# B&R Automation Studio project Soiled_PLC (part 3)

#### 7_sdc2Cyclic.ab
```automation-basic
PROGRAM _CYCLIC
	(* cyclic program *)

;Sequence 7 - Discharger 2 D[907]

;-----------------------------------------
;Revision 1.00 19/12/2005 D.J. First Issue
;-----------------------------------------

DischargerEnable 		= ((D[15] > 0) AND NOT Std.HaltSys)

;I_BagAtBuffer			= X[6].X07
I_OpenBag				= X[1].X05              ;CAN[2].DropLoad OR TestDrop
I_LoadDropped			= X[1].X06             ;CAN[2].LoadDropped OR TestDropped
I_BagAtBuffer			= X[1].X02 OR TestBuffer
I_BagAtDischarger		= X[1].X03 OR TestAtDisch
I_BagEmpty			  	= TRUE

I_BagAtEmptyBuffer		= FALSE ;X[6].X13
O_EmptyBagBufferOpen	= FALSE ;Y[6].Y13

O_BagReady				= FALSE
O_OpenBuffer 			= FALSE
O_Steadys				= FALSE
O_Closer				= FALSE
O_OpenBag				= FALSE
O_OpenStop				= FALSE

;Alarm
Alarm[10].Name 			= almNoAlarm ;Clear sequence alarm name
Alarm[10].Bag 			= 80
Alarm[10].Beacon		= TRUE
Alarm[10].Extra			= 0
Alarm[10].Time			= 3000

;Setup Sequence
STEP = D[910]
;Setup Pulse contact
PLS = (STEP <> LASTSTEP)
LASTSTEP = STEP

;Step 0 - Disabled
IF (STEP = 0) THEN
	;Disabled
ENDIF

;Check Status - Bag settled at buffer, no bag at discharger, bag at buffer on screen and no bag at discharger on the screen
TON_10ms(I_BagAtBuffer,300,SettledAtBuffer,SettledAtBufferET)
IF (STEP = 1) THEN
	IF (NOT I_BagAtDischarger AND  (Bag[80].Cat = 0) AND NOT Std.HaltSys AND DischargerEnable AND SettledAtBuffer) THEN
		Request.DC[2] = TRUE
		D[910] = 2
	ENDIF
	IF I_BagAtDischarger THEN
		;D[907] = 2
	ENDIF
	IF (Bag[80].Cat > 0) THEN
		Alarm[10].Name = almBagDataError
	ELSE IF I_BagAtDischarger THEN
		Alarm[10].Name = almSwitchFault
	ELSE IF (Bag[80].Cat > 0) AND NOT I_BagAtBuffer THEN
		Alarm[10].Name 	= almBagNotAtProx
		Alarm[10].Bag	= 80
	ELSE IF (Bag[80].Cat = 0) AND I_BagAtBuffer AND DischargerEnable  THEN
		Alarm[10].Name 	= almBagNotShownOnScreen
		Alarm[10].Bag	= 80
	ENDIF
ENDIF

;Wait for bag in discharger
IF (STEP = 2) THEN
	O_OpenBuffer 	= TRUE
	IF I_BagAtDischarger THEN
		D[910] = 3
	ENDIF
	Alarm[10].Name = almNoAlarm ;almBagNotArrived
ENDIF

;Let bag settle in discharger
TON_10ms(((STEP = 3) AND I_BagAtDischarger),1000,SettledAtDischarger,SettledAtDischargerET)
IF (STEP = 3) THEN
	IF (Bag[80].Cat = 0) AND (Bag[81].Cat > 0) THEN
		Bag[80] = Bag[81]
		Bag[81] = Bag[0]
	ENDIF
	IF SettledAtDischarger THEN
		D[910] = 4
	ENDIF
	Alarm[10].Name = almBagNotSettled
ENDIF

;Allow steadys to move down
TON_10ms((STEP = 4),400,SteadysDown,SteadysDownET)
IF (STEP = 4) THEN
	IF SteadysDown THEN
		D[910] = 5
	ENDIF
	IF (Bag[80].Cat = Std.MaxCats) THEN
		D[910] = 8
	ENDIF
ENDIF

;Steady cylinders on from steps 4 - 9
O_Steadys = ((STEP >= 4) AND (STEP <= 9))

;Bag opener on from step 5 - 8
O_OpenBag = ((STEP >= 6) AND (STEP <= 8))

CodeStep  = ((STEP >= 4) AND (STEP <= 5))

;Wash Codes
IF CodeStep THEN

	Weight = Bag[80].Wgt

	;round up weight to give to wash machine
	Remainder = SINT(Bag[80].Wgt MOD 10)
	IF (Remainder > 4) THEN
		WgtRound = (Weight + 10)
	ELSE
		WgtRound = Weight
	ENDIF
ELSE
ENDIF

;Bag Ready to Washing Machine
IF (STEP = 5) THEN
	O_BagReady = TRUE

	IF I_OpenBag OR TestDischarger THEN
		D[910] = 6
	ENDIF
ELSE

ENDIF

;Set LoadDropped to False
IF (STEP <> 6) THEN
	LoadDropped = FALSE
ENDIF

;Open Bag Until LoadDropped recieved and has been open for 6 seconds
TON_10ms((STEP = 6),600,MinOpen,MinOpenET) ;ET means Elapsed Time
TON_10ms((STEP = 6) AND NOT I_DischargerBagEmpty ,100,BagEmpty,BagEmptyET)

IF (STEP = 6) THEN

	;IF I_LoadDropped  OR TestDischarger THEN

		LoadDropped = TRUE
	;ENDIF

	IF (LoadDropped AND MinOpen) THEN
		;Write Report
		;------------

	ENDIF
	IF (LoadDropped AND MinOpen ) THEN
		IF (ReportUnloading[5].Cat = 0) THEN
			ReportUnloading[5].Cat = UINT(Bag[80].Cat)	;Category
			ReportUnloading[5].Cus = Bag[80].Cus		;Customer
			ReportUnloading[5].Wgt = Bag[80].Wgt		;Weight
			ReportUnloading[5].Cnt = 0					;Count
			ReportUnloading[5].Stn = 0					;Station
			ReportUnloading[5].Mcn = 5					;Machine
		ENDIF
		D[910] = 7
	ENDIF
	Alarm[10].Time			= 600
	Alarm[10].Name = almLoadNotDropped
	ELSE
	LoadDropped = FALSE
ENDIF

;Change display to empty bag
IF (STEP = 7) THEN
	IF ((NOT I_OpenBag  AND I_BagEmpty) OR TestDrop) THEN
		Bag[80].Prg 	= Std.MaxProg
		Bag[80].Cat 	= Std.MaxCats
		Bag[80].Cus 	= Std.MaxCust

		D[910] 			= 8
	ENDIF
	Alarm[10].Name = almGeneralSequence
ENDIF

;Allow steadys to go up
TON_10ms((STEP = 8),400,SteadyUp,SteadyUpET)
IF (STEP = 8) THEN
	IF SteadyUp THEN
		D[910] = 9
	ENDIF
ENDIF

;Request empty bag release
IF (STEP = 9) THEN

	IF Line[32].Clear THEN
		C[32]  = 0
		D[910] = 10
	ENDIF
ENDIF

;Open buffer stop - unitl bag out
IF (STEP = 10) THEN
	O_OpenStop = TRUE
	Bag[80].Cat = 0
	Bag[80].Cus = 0
	Bag[80].Wgt = 0
	IF Line[32].Trip THEN
		D[910] = 1
	ENDIF
	Alarm[10].Name = almBagNotReleased
ENDIF

;Alarms
TimerAlarm.IN 	= NOT PLS AND (Alarm[10].Name > 0)
TimerAlarm.PT 	= Alarm[10].Time
TimerAlarm FUB TON_10ms()
Alarm[10].On 	= TimerAlarm.Q
Alarm[10].ET 	= TimerAlarm.ET

;Outputs
Y[1].Y02 = O_OpenBuffer
Y[1].Y04= O_Steadys
Y[1].Y06 = O_OpenBag
Y[1].Y03 = O_OpenStop
Y[1].Y05 = O_BagReady
END_PROGRAM
```

### Program Logical/Sequences/10ms/11_sdc6 (IEC) - * SDC2 Machine 2 CAN

#### 7_sdc2Cyclic.ab
```automation-basic
PROGRAM _CYCLIC
	(* cyclic program *)

;Sequence 7 - Discharger 2 D[907]

;-----------------------------------------
;Revision 1.00 19/12/2005 D.J. First Issue
;-----------------------------------------

DischargerEnable 		= ((D[26] > 0) AND NOT Std.HaltSys)

;I_BagAtBuffer			= X[6].X07
I_OpenBag				= X[1].X11
I_LoadDropped			= X[1].X12
I_BagAtBuffer			= X[1].X08 OR TestBuffer
I_BagAtDischarger		= X[1].X09 OR TestAtDisch
I_BagEmpty			  	= TRUE
I_BagOut                  = X[1].X10

RequestRel.DC[6]                   = FALSE

O_BagReady				= FALSE
O_OpenBuffer 			= FALSE
O_Steadys				= FALSE
O_Closer				= FALSE
O_OpenBag				= FALSE
O_OpenStop				= FALSE

;Alarm
Alarm[11].Name 			= almNoAlarm ;Clear sequence alarm name
Alarm[11].Bag 			= 85
Alarm[11].Beacon			= TRUE
Alarm[11].Extra			= 0
Alarm[11].Time			= 3000

;Setup Sequence
STEP = D[911]
;Setup Pulse contact
PLS = (STEP <> LASTSTEP)
LASTSTEP = STEP

;Step 0 - Disabled
IF (STEP = 0) THEN
	;Disabled
ENDIF

;Check Status - Bag settled at buffer, no bag at discharger, bag at buffer on screen and no bag at discharger on the screen
TON_10ms(I_BagAtBuffer,300,SettledAtBuffer,SettledAtBufferET)
IF (STEP = 1) THEN
	IF (NOT I_BagAtDischarger AND  (Bag[85].Cat = 0) AND NOT Std.HaltSys AND DischargerEnable AND SettledAtBuffer) THEN

		D[911] = 2
	ENDIF
	IF I_BagAtDischarger THEN
		;D[907] = 2
	ENDIF
	IF (Bag[85].Cat > 0) THEN
		Alarm[11].Name = almBagDataError
	ELSE IF I_BagAtDischarger THEN
		Alarm[11].Name = almSwitchFault
	ELSE IF (Bag[85].Cat > 0) AND NOT I_BagAtBuffer THEN
		Alarm[11].Name 	= almBagNotAtProx
		Alarm[11].Bag	= 85
	ELSE IF (Bag[85].Cat = 0) AND I_BagAtBuffer AND DischargerEnable  THEN
		Alarm[11].Name 	= almBagNotShownOnScreen
		Alarm[11].Bag	= 85
	ENDIF
ENDIF

;Wait for bag in discharger
IF (STEP = 2) THEN
	O_OpenBuffer 	= TRUE
	IF I_BagAtDischarger THEN
		D[911] = 3
	ENDIF
	Alarm[11].Name = almNoAlarm ;almBagNotArrived
ENDIF

;Let bag settle in discharger
TON_10ms(((STEP = 3) AND I_BagAtDischarger),1000,SettledAtDischarger,SettledAtDischargerET)
IF (STEP = 3) THEN
	IF (Bag[85].Cat = 0) AND (Bag[86].Cat > 0) THEN
		Bag[85] = Bag[86]
		Bag[86] = Bag[0]
	ENDIF
	IF SettledAtDischarger THEN
		D[911] = 4
	ENDIF
	Alarm[11].Name = almBagNotSettled
ENDIF

;Allow steadys to move down
TON_10ms((STEP = 4),400,SteadysDown,SteadysDownET)
IF (STEP = 4) THEN
	IF SteadysDown THEN
		D[911] = 5
	ENDIF
	IF (Bag[85].Cat = Std.MaxCats) THEN
		D[911] = 8
	ENDIF
ENDIF

;Steady cylinders on from steps 4 - 9
O_Steadys = ((STEP >= 4) AND (STEP <= 7))

;Bag opener on from step 5 - 8
O_OpenBag = ((STEP >= 6) AND (STEP <= 7))

CodeStep  = ((STEP >= 4) AND (STEP <= 5))

;Wash Codes
IF CodeStep THEN

	Weight = Bag[85].Wgt

	;round up weight to give to wash machine
	Remainder = SINT(Bag[85].Wgt MOD 10)
	IF (Remainder > 4) THEN
		WgtRound = (Weight + 10)
	ELSE
		WgtRound = Weight
	ENDIF

	;WashCodes
	;if Below the Machine limit of 99 and no WashCode has been entered then send the Category

ELSE

ENDIF

;Bag Ready to Washing Machine
IF (STEP = 5) THEN
	O_BagReady		= TRUE

	IF I_OpenBag OR TestDischarger THEN
		D[911] = 6
	ENDIF
ELSE
	O_BagReady		= FALSE
ENDIF

;Set LoadDropped to False
IF (STEP <> 6) THEN
	LoadDropped = FALSE
ENDIF

;Open Bag Until LoadDropped recieved and has been open for 6 seconds
TON_10ms((STEP = 6),600,MinOpen,MinOpenET) ;ET means Elapsed Time
TON_10ms((STEP = 6) AND NOT I_DischargerBagEmpty ,100,BagEmpty,BagEmptyET)

IF (STEP = 6) THEN

	IF I_LoadDropped  OR TestDischarger THEN

		LoadDropped = TRUE
	ENDIF

	IF (LoadDropped AND MinOpen) THEN
		;Write Report
		;------------

	ENDIF
	IF (LoadDropped AND MinOpen ) THEN
		IF (ReportUnloading[6].Cat = 0) THEN
			ReportUnloading[6].Cat = UINT(Bag[85].Cat)	;Category
			ReportUnloading[6].Cus = Bag[85].Cus		;Customer
			ReportUnloading[6].Wgt = Bag[85].Wgt		;Weight
			ReportUnloading[6].Cnt = 0					;Count
			ReportUnloading[6].Stn = 0					;Station
			ReportUnloading[6].Mcn = 6					;Machine
		ENDIF
		D[911] = 7
	ENDIF
	Alarm[11].Time			= 600
	Alarm[11].Name = almLoadNotDropped
	ELSE
	LoadDropped = FALSE
ENDIF

;Change display to empty bag
IF (STEP = 7) THEN
	IF ((NOT I_OpenBag  AND I_BagEmpty) OR TestDrop) THEN
		Bag[85].Prg 	= Std.MaxProg
		Bag[85].Cat 	= Std.MaxCats
		Bag[85].Cus 	= Std.MaxCust

		D[911] 			= 8
	ENDIF
	Alarm[11].Name = almGeneralSequence
ENDIF

;Allow steadys to go up
TON_10ms((STEP = 8),400,SteadyUp,SteadyUpET)
IF (STEP = 8) THEN
	IF SteadyUp THEN
		D[911] = 9
	ENDIF
ENDIF

;Request empty bag release
IF (STEP = 9) THEN
	RequestRel.DC[6] = TRUE
	IF Enable.DCEmptyRelease[6] THEN
		;C[32]  = 0
		D[911] = 10
	ENDIF
ENDIF

;Open buffer stop - unitl bag out
IF (STEP = 10) THEN
	O_OpenStop = TRUE
	Bag[85].Cat = 0
	Bag[85].Cus = 0
	Bag[85].Wgt = 0
	IF NOT Enable.DCEmptyRelease[6] OR I_BagOut THEN
		D[911] = 1
	ENDIF
	Alarm[11].Name = almBagNotReleased
ENDIF

;Alarms
TimerAlarm.IN 	= NOT PLS AND (Alarm[11].Name > 0)
TimerAlarm.PT 	= Alarm[11].Time
TimerAlarm FUB TON_10ms()
Alarm[11].On 	= TimerAlarm.Q
Alarm[11].ET 	= TimerAlarm.ET

;Outputs
Y[1].Y08 = O_OpenBuffer
Y[1].Y10 = O_Steadys
Y[1].Y12 = O_OpenBag
Y[1].Y09 = O_OpenStop
Y[1].Y11 = O_BagReady
END_PROGRAM
```

### Program Logical/Sequences/10ms/12_sdc7 (IEC) - * SDC2 Machine 2 CAN

#### 7_sdc2Cyclic.ab
```automation-basic
PROGRAM _CYCLIC
	(* cyclic program *)

;Sequence 7 - Discharger 2 D[907]

;-----------------------------------------
;Revision 1.00 19/12/2005 D.J. First Issue
;-----------------------------------------

DischargerEnable 		= ((D[27] > 0) AND NOT Std.HaltSys)

;I_BagAtBuffer			= X[6].X07
I_OpenBag				= X[2].X01 ;0CAN[2].DropLoad OR TestDrop
I_LoadDropped			= X[2].X02
I_BagAtBuffer			= X[1].X14 OR TestBuffer
I_BagAtDischarger		= X[1].X15 OR TestAtDisch
I_BagEmpty			  	= TRUE
I_BagOut                  = X[1].X16

I_BagAtEmptyBuffer		= FALSE ;X[6].X13
O_EmptyBagBufferOpen	= FALSE ;Y[6].Y13

O_BagReady				= FALSE
O_OpenBuffer 			= FALSE
O_Steadys				= FALSE
O_Closer				= FALSE
O_OpenBag				= FALSE
O_OpenStop				= FALSE

;Alarm
Alarm[12].Name 			= almNoAlarm ;Clear sequence alarm name
Alarm[12].Bag 			= 90
Alarm[12].Beacon		= TRUE
Alarm[12].Extra			= 0
Alarm[12].Time			= 3000

;Setup Sequence
STEP = D[912]
;Setup Pulse contact
PLS = (STEP <> LASTSTEP)
LASTSTEP = STEP

;Step 0 - Disabled
IF (STEP = 0) THEN
	;Disabled
ENDIF

;Check Status - Bag settled at buffer, no bag at discharger, bag at buffer on screen and no bag at discharger on the screen
TON_10ms(I_BagAtBuffer,300,SettledAtBuffer,SettledAtBufferET)
IF (STEP = 1) THEN
	IF (NOT I_BagAtDischarger AND  (Bag[90].Cat = 0) AND NOT Std.HaltSys AND DischargerEnable AND SettledAtBuffer) THEN

		D[912] = 2
	ENDIF
	IF I_BagAtDischarger THEN
		;D[907] = 2
	ENDIF
	IF (Bag[90].Cat > 0) THEN
		Alarm[12].Name = almBagDataError
	ELSE IF I_BagAtDischarger THEN
		Alarm[12].Name = almSwitchFault
	ELSE IF (Bag[91].Cat > 0) AND NOT I_BagAtBuffer THEN
		Alarm[12].Name 	= almBagNotAtProx
		Alarm[12].Bag	= 91
	ELSE IF (Bag[91].Cat = 0) AND I_BagAtBuffer AND DischargerEnable  THEN
		Alarm[12].Name 	= almBagNotShownOnScreen
		Alarm[12].Bag	= 91
	ENDIF
ENDIF

;Wait for bag in discharger
IF (STEP = 2) THEN
	O_OpenBuffer 	= TRUE
	IF I_BagAtDischarger THEN
		D[912] = 3
	ENDIF
	Alarm[12].Name = almNoAlarm ;almBagNotArrived
ENDIF

;Let bag settle in discharger
TON_10ms(((STEP = 3) AND I_BagAtDischarger),1000,SettledAtDischarger,SettledAtDischargerET)
IF (STEP = 3) THEN
	IF (Bag[90].Cat = 0) AND (Bag[91].Cat > 0) THEN
		Bag[90] = Bag[91]
		Bag[91] = Bag[0]
	ENDIF
	IF SettledAtDischarger THEN
		D[912] = 4
	ENDIF
	Alarm[12].Name = almBagNotSettled
ENDIF

;Allow steadys to move down
TON_10ms((STEP = 4),400,SteadysDown,SteadysDownET)
IF (STEP = 4) THEN
	IF SteadysDown THEN
		D[912] = 5
	ENDIF
	IF (Bag[90].Cat = Std.MaxCats) THEN
		D[912] = 8
	ENDIF
ENDIF

;Steady cylinders on from steps 4 - 9
O_Steadys = ((STEP >= 4) AND (STEP <= 9))

;Bag opener on from step 5 - 8
O_OpenBag = ((STEP >= 6) AND (STEP <= 8))

CodeStep  = ((STEP >= 4) AND (STEP <= 5))

;Wash Codes
IF CodeStep THEN

	Weight = Bag[90].Wgt

	;round up weight to give to wash machine
	Remainder = SINT(Bag[90].Wgt MOD 10)
	IF (Remainder > 4) THEN
		WgtRound = (Weight + 10)
	ELSE
		WgtRound = Weight
	ENDIF

ELSE

ENDIF

;Bag Ready to Washing Machine
IF (STEP = 5) THEN
	O_BagReady 		= TRUE

	IF I_OpenBag OR TestDischarger THEN
		D[912] = 6
	ENDIF
ELSE

ENDIF

;Set LoadDropped to False
IF (STEP <> 6) THEN
	LoadDropped = FALSE
ENDIF

;Open Bag Until LoadDropped recieved and has been open for 6 seconds
TON_10ms((STEP = 6),600,MinOpen,MinOpenET) ;ET means Elapsed Time
TON_10ms((STEP = 6) AND NOT I_DischargerBagEmpty ,100,BagEmpty,BagEmptyET)

IF (STEP = 6) THEN

	;IF I_LoadDropped  OR TestDischarger THEN

		LoadDropped = TRUE
	;ENDIF

	IF (LoadDropped AND MinOpen) THEN
		;Write Report
		;------------

	ENDIF
	IF (LoadDropped AND MinOpen ) THEN
		IF (ReportUnloading[2].Cat = 0) THEN
			ReportUnloading[2].Cat = UINT(Bag[90].Cat)	;Category
			ReportUnloading[2].Cus = Bag[90].Cus		;Customer
			ReportUnloading[2].Wgt = Bag[90].Wgt		;Weight
			ReportUnloading[2].Cnt = 0					;Count
			ReportUnloading[2].Stn = 0					;Station
			ReportUnloading[2].Mcn = 7					;Machine
		ENDIF
		D[912] = 7
	ENDIF
	Alarm[12].Time			= 600
	Alarm[12].Name = almLoadNotDropped
	ELSE
	LoadDropped = FALSE
ENDIF

;Change display to empty bag
IF (STEP = 7) THEN
	IF ((NOT I_OpenBag  AND I_BagEmpty) OR TestDrop) THEN
		Bag[90].Prg 	= Std.MaxProg
		Bag[90].Cat 	= Std.MaxCats
		Bag[90].Cus 	= Std.MaxCust

		D[912] 			= 8
	ENDIF
	Alarm[12].Name = almGeneralSequence
ENDIF

;Allow steadys to go up
TON_10ms((STEP = 8),400,SteadyUp,SteadyUpET)
IF (STEP = 8) THEN
	IF SteadyUp AND NOT Enable.DCEmptyRelease[7] THEN
		D[912] = 9
	ENDIF
	IF Enable.DCEmptyRelease[7]  THEN
		Alarm[12].Time			= 600
		Alarm[12].Name = almSwitchFault
	ENDIF
ENDIF

;Request empty bag release
IF (STEP = 9) THEN
	RequestRel.DC[7] = TRUE
	IF Enable.DCEmptyRelease[7] THEN
		;C[32]  = 0
		D[912] = 10
	ENDIF
	ELSE
	RequestRel.DC[7] = FALSE
ENDIF

;Open buffer stop - unitl bag out
IF (STEP = 10) THEN
	O_OpenStop = TRUE
	Bag[90].Cat = 0
	Bag[90].Cus = 0
	Bag[90].Wgt = 0
	IF NOT Enable.DCEmptyRelease[7]  OR I_BagOut THEN
		D[912] = 1
	ENDIF
	Alarm[12].Name = almBagNotReleased
ENDIF

;Alarms
TimerAlarm.IN 	= NOT PLS AND (Alarm[12].Name > 0)
TimerAlarm.PT 	= Alarm[12].Time
TimerAlarm FUB TON_10ms()
Alarm[12].On 	= TimerAlarm.Q
Alarm[12].ET 	= TimerAlarm.ET

;Outputs
Y[1].Y14 = O_OpenBuffer
Y[1].Y16 = O_Steadys
Y[2].Y02 = O_OpenBag
Y[1].Y15 = O_OpenStop
Y[2].Y01= O_BagReady
END_PROGRAM
```

### Program Logical/Sequences/10ms/13_sdc8 (IEC) - * SDC2 Machine 2 CAN

#### 7_sdc2.var
```iecst
VAR RETAIN
	STEP : UINT;
	PLS : BOOL;
	LASTSTEP : UINT;
	SteadyUp : BOOL;
	CloserUpET : TIME;
	SteadysDown : BOOL;
	SteadysDownET : TIME;
	LoadDropped : BOOL;
	SteadyUpET : TIME;
	CloserDownET : TIME;
	SettledAtDischargerET : TIME;
	MinOpenET : TIME;
	SettledAtDischarger : BOOL;
	CloserDown : BOOL;
	MinOpen : BOOL;
	CloserUp : BOOL;
	SettledAtBuffer : BOOL;
	SettledAtBufferET : TIME;
	I_BagAtBuffer : BOOL;
	O_OpenStop : BOOL;
	O_OpenBag : BOOL;
	O_Steadys : BOOL;
	O_OpenBuffer : BOOL;
	O_Closer : BOOL;
	I_BagAtDischarger : BOOL;
	I_OpenBag : BOOL;
	I_LoadDropped : BOOL;
	TestDrop : BOOL;
END_VAR
VAR
	DischargerEnable : BOOL;
	TestDischarger : BOOL;
	I_BagEmpty : BOOL;
	O_BagReady : BOOL;
	WgtRound : UINT;
	TimerAlarm : TON_10ms;
	I_BagReleased : BOOL;
	O_EmptyBagBufferOpen : BOOL;
	I_BagAtEmptyBuffer : BOOL;
	Remainder : UINT;
	CodeStep : BOOL;
	I_DischargerBagEmpty : BOOL;
	BagEmpty : BOOL;
	BagEmptyET : TIME;
	BCD_BIN_CAT : BCD_BIN_OUTPUT;
	BCD_BIN_CUS : BCD_BIN_OUTPUT;
	BCD_BIN_WGT : BCD_BIN_OUTPUT;
	TestDropped : BOOL;
	TestBuffer : BOOL;
	TestAtDisch : BOOL;
	Weight : UINT;
	I_BagOut : BOOL;
END_VAR
```

#### 7_sdc2Cyclic.ab
```automation-basic
PROGRAM _CYCLIC
	(* cyclic program *)

;Sequence 7 - Discharger 2 D[907]

;-----------------------------------------
;Revision 1.00 19/12/2005 D.J. First Issue
;-----------------------------------------

DischargerEnable 		= ((D[28] > 0) AND NOT Std.HaltSys)

;I_BagAtBuffer			= X[6].X07
I_OpenBag				= X[2].X07
I_LoadDropped			= X[2].X08
I_BagAtBuffer			= X[2].X04 OR TestBuffer
I_BagAtDischarger		= X[2].X05 OR TestAtDisch
I_BagEmpty			  	= TRUE
I_BagOut                  = X[2].X06

O_BagReady				= FALSE
O_OpenBuffer 			= FALSE
O_Steadys				= FALSE
O_Closer				= FALSE
O_OpenBag				= FALSE
O_OpenStop				= FALSE
RequestRel.DC[8]      = FALSE

;Alarm
Alarm[13].Name 			= almNoAlarm ;Clear sequence alarm name
Alarm[13].Bag 			= 95
Alarm[13].Beacon		= TRUE
Alarm[13].Extra			= 0
Alarm[13].Time			= 3000

;Setup Sequence
STEP = D[913]
;Setup Pulse contact
PLS = (STEP <> LASTSTEP)
LASTSTEP = STEP

;Step 0 - Disabled
IF (STEP = 0) THEN
	;Disabled
ENDIF

;Check Status - Bag settled at buffer, no bag at discharger, bag at buffer on screen and no bag at discharger on the screen
TON_10ms(I_BagAtBuffer,300,SettledAtBuffer,SettledAtBufferET)
IF (STEP = 1) THEN
	IF (NOT I_BagAtDischarger AND  (Bag[95].Cat = 0) AND NOT Std.HaltSys AND DischargerEnable AND SettledAtBuffer) THEN
		Request.DC[2] = TRUE
		D[913] = 2
	ENDIF
	IF I_BagAtDischarger THEN
		;D[907] = 2
	ENDIF
	IF (Bag[95].Cat > 0) THEN
		Alarm[13].Name = almBagDataError
	ELSE IF I_BagAtDischarger THEN
		Alarm[13].Name = almSwitchFault
	ELSE IF (Bag[96].Cat > 0) AND NOT I_BagAtBuffer THEN
		Alarm[13].Name 	= almBagNotAtProx
		Alarm[13].Bag	= 96
	ELSE IF (Bag[96].Cat = 0) AND I_BagAtBuffer AND DischargerEnable  THEN
		Alarm[13].Name 	= almBagNotShownOnScreen
		Alarm[13].Bag	= 96
	ENDIF
ENDIF

;Wait for bag in discharger
IF (STEP = 2) THEN
	O_OpenBuffer 	= TRUE
	IF I_BagAtDischarger THEN
		D[913] = 3
	ENDIF
	Alarm[13].Name = almNoAlarm ;almBagNotArrived
ENDIF

;Let bag settle in discharger
TON_10ms(((STEP = 3) AND I_BagAtDischarger),1000,SettledAtDischarger,SettledAtDischargerET)
IF (STEP = 3) THEN
	IF (Bag[95].Cat = 0) AND (Bag[96].Cat > 0) THEN
		Bag[95] = Bag[96]
		Bag[96] = Bag[0]
	ENDIF
	IF SettledAtDischarger THEN
		D[913] = 4
	ENDIF
	Alarm[13].Name = almBagNotSettled
ENDIF

;Allow steadys to move down
TON_10ms((STEP = 4),400,SteadysDown,SteadysDownET)
IF (STEP = 4) THEN
	IF SteadysDown THEN
		D[913] = 5
	ENDIF
	IF (Bag[95].Cat = Std.MaxCats) THEN
		D[913] = 8
	ENDIF
ENDIF

;Steady cylinders on from steps 4 - 9
O_Steadys = ((STEP >= 4) AND (STEP <= 9))

;Bag opener on from step 5 - 8
O_OpenBag = ((STEP >= 6) AND (STEP <= 8))

;CodeStep  = ((STEP >= 4) AND (STEP <= 5))

;Wash Codes
IF CodeStep THEN

	Weight = Bag[188].Wgt

	;round up weight to give to wash machine
	Remainder = SINT(Bag[188].Wgt MOD 10)
	IF (Remainder > 4) THEN
		WgtRound = (Weight + 10)
	ELSE
		WgtRound = Weight
	ENDIF

	;WashCodes
	;if Below the Machine limit of 99 and no WashCode has been entered then send the Category

	CAN[2].Category 	= Bag[188].Cat
	CAN[2].Customer 	= Bag[188].Cus
	CAN[2].Weight   	= (WgtRound / 10) ;rounded up weight divide by 10
	;CAN[1].DoubleLoad 	= (Batch > 0)
ELSE
	;CAN[2].Category 	= 0
	;CAN[2].Customer 	= 0
	;CAN[2].Weight   	= 0
	;CAN[1].DoubleLoad 	= FALSE

ENDIF

;Bag Ready to Washing Machine
IF (STEP = 5) THEN
	O_BagReady	 		= TRUE

	IF I_OpenBag OR TestDischarger THEN
		D[913] = 6
	ENDIF
ELSE
	O_BagReady	 = FALSE
ENDIF

;Set LoadDropped to False
IF (STEP <> 6) THEN
	LoadDropped = FALSE
ENDIF

;Open Bag Until LoadDropped recieved and has been open for 6 seconds
TON_10ms((STEP = 6),600,MinOpen,MinOpenET) ;ET means Elapsed Time
TON_10ms((STEP = 6) AND NOT I_DischargerBagEmpty ,100,BagEmpty,BagEmptyET)

IF (STEP = 6) THEN

	;IF I_LoadDropped  OR TestDischarger THEN

		LoadDropped = TRUE
	;ENDIF

	IF (LoadDropped AND MinOpen) THEN
		;Write Report
		;------------

	ENDIF
	IF (LoadDropped AND MinOpen ) THEN
		IF (ReportUnloading[8].Cat = 0) THEN
			ReportUnloading[8].Cat = UINT(Bag[95].Cat)	;Category
			ReportUnloading[8].Cus = Bag[95].Cus		;Customer
			ReportUnloading[8].Wgt = Bag[95].Wgt		;Weight
			ReportUnloading[8].Cnt = 0					;Count
			ReportUnloading[8].Stn = 0					;Station
			ReportUnloading[8].Mcn = 8					;Machine
		ENDIF
		D[913] = 7
	ENDIF
	Alarm[13].Time			= 600
	Alarm[13].Name = almLoadNotDropped
	ELSE
	LoadDropped = FALSE
ENDIF

;Change display to empty bag
IF (STEP = 7) THEN
	IF ((NOT I_OpenBag  AND I_BagEmpty) OR TestDrop) THEN
		Bag[95].Prg 	= Std.MaxProg
		Bag[95].Cat 	= Std.MaxCats
		Bag[95].Cus 	= Std.MaxCust

		D[913] 			= 8
	ENDIF
	Alarm[13].Name = almGeneralSequence
ENDIF

;Allow steadys to go up
TON_10ms((STEP = 8),400,SteadyUp,SteadyUpET)
IF (STEP = 8) THEN
	IF SteadyUp AND NOT Enable.DCEmptyRelease[8]  THEN
		D[913] = 9
	ENDIF
	IF Enable.DCEmptyRelease[8] THEN
		Alarm[13].Name = almSwitchFault
	ENDIF
ENDIF

;Request empty bag release
IF (STEP = 9) THEN
	RequestRel.DC[8] = TRUE
	IF Enable.DCEmptyRelease[8] THEN
		;C[32]  = 0
		D[913] = 10
	ENDIF
ENDIF

;Open buffer stop - unitl bag out
IF (STEP = 10) THEN
	O_OpenStop = TRUE
	Bag[95].Cat = 0
	Bag[95].Cus = 0
	Bag[95].Wgt = 0
	IF I_BagOut  OR (Enable.DCEmptyRelease[8]= FALSE) THEN
		D[913] = 1
	ENDIF
	Alarm[13].Name = almBagNotReleased
ENDIF

;Alarms
TimerAlarm.IN 	= NOT PLS AND (Alarm[13].Name > 0)
TimerAlarm.PT 	= Alarm[13].Time
TimerAlarm FUB TON_10ms()
Alarm[13].On 	= TimerAlarm.Q
Alarm[13].ET 	= TimerAlarm.ET

;Outputs
Y[2].Y04 = O_OpenBuffer
Y[2].Y06 = O_Steadys
Y[2].Y08 = O_OpenBag
Y[2].Y05 = O_OpenStop
Y[2].Y07 = O_BagReady
END_PROGRAM
```

### Program Logical/Sequences/10ms/14_sdc9 (IEC) - * SDC2 Machine 2 CAN

#### 7_sdc2Cyclic.ab
```automation-basic
PROGRAM _CYCLIC
	(* cyclic program *)

;Sequence 7 - Discharger 2 D[907]

;-----------------------------------------
;Revision 1.00 19/12/2005 D.J. First Issue
;-----------------------------------------

DischargerEnable 		= ((D[29] > 0) AND NOT Std.HaltSys)

;I_BagAtBuffer			= X[6].X07
I_OpenBag				= X[2].X13
I_LoadDropped			= X[2].X14
I_BagAtBuffer			= X[2].X10 OR TestBuffer
I_BagAtDischarger		= X[2].X11 OR TestAtDisch
I_BagEmpty			  	= TRUE

I_BagAtEmptyBuffer		= FALSE ;X[6].X13
O_EmptyBagBufferOpen	= FALSE ;Y[6].Y13

O_BagReady				          = FALSE
O_OpenBuffer 			            = FALSE
O_Steadys				             = FALSE
O_Closer				               = FALSE
O_OpenBag			            	= FALSE
O_OpenStop				           = FALSE
Request.DCEmptyRelease[9] = FALSE

;Alarm
Alarm[14].Name 			= almNoAlarm ;Clear sequence alarm name
Alarm[14].Bag 			= 100
Alarm[14].Beacon		= TRUE
Alarm[14].Extra			= 0
Alarm[14].Time			= 3000

;Setup Sequence
STEP = D[914]
;Setup Pulse contact
PLS = (STEP <> LASTSTEP)
LASTSTEP = STEP

;Step 0 - Disabled
IF (STEP = 0) THEN
	;Disabled
ENDIF

;Check Status - Bag settled at buffer, no bag at discharger, bag at buffer on screen and no bag at discharger on the screen
TON_10ms(I_BagAtBuffer,300,SettledAtBuffer,SettledAtBufferET)
IF (STEP = 1) THEN
	IF (NOT I_BagAtDischarger AND  (Bag[100].Cat = 0) AND NOT Std.HaltSys AND DischargerEnable AND SettledAtBuffer) THEN

		D[914] = 2
	ENDIF
	IF I_BagAtDischarger THEN
		;D[907] = 2
	ENDIF
	IF (Bag[100].Cat > 0) THEN
		Alarm[14].Name = almBagDataError
	ELSE IF I_BagAtDischarger THEN
		Alarm[14].Name = almSwitchFault
	ELSE IF (Bag[101].Cat > 0) AND NOT I_BagAtBuffer THEN
		Alarm[14].Name 	= almBagNotAtProx
		Alarm[14].Bag	= 100
	ELSE IF (Bag[101].Cat = 0) AND I_BagAtBuffer AND DischargerEnable  THEN
		Alarm[14].Name 	= almBagNotShownOnScreen
		Alarm[14].Bag	= 100
	ENDIF
ENDIF

;Wait for bag in discharger
IF (STEP = 2) THEN
	O_OpenBuffer 	= TRUE
	IF I_BagAtDischarger THEN
		D[914] = 3
	ENDIF
	Alarm[14].Name = almNoAlarm ;almBagNotArrived
ENDIF

;Let bag settle in discharger
TON_10ms(((STEP = 3) AND I_BagAtDischarger),1000,SettledAtDischarger,SettledAtDischargerET)
IF (STEP = 3) THEN
	IF (Bag[100].Cat = 0) AND (Bag[101].Cat > 0) THEN
		Bag[100] = Bag[101]
		Bag[101] = Bag[0]
	ENDIF
	IF SettledAtDischarger THEN
		D[914] = 4
	ENDIF
	Alarm[14].Name = almBagNotSettled
ENDIF

;Allow steadys to move down
TON_10ms((STEP = 4),400,SteadysDown,SteadysDownET)
IF (STEP = 4) THEN
	IF SteadysDown THEN
		D[914] = 5
	ENDIF
	IF (Bag[100].Cat = Std.MaxCats) THEN
		D[914] = 8
	ENDIF
ENDIF

;Steady cylinders on from steps 4 - 9
O_Steadys = ((STEP >= 4) AND (STEP <= 9))

;Bag opener on from step 5 - 8
O_OpenBag = ((STEP >= 6) AND (STEP <= 8))

;CodeStep  = ((STEP >= 4) AND (STEP <= 5))

;Wash Codes
IF CodeStep THEN

	Weight = Bag[188].Wgt

	;round up weight to give to wash machine
	Remainder = SINT(Bag[188].Wgt MOD 10)
	IF (Remainder > 4) THEN
		WgtRound = (Weight + 10)
	ELSE
		WgtRound = Weight
	ENDIF

	;WashCodes
	;if Below the Machine limit of 99 and no WashCode has been entered then send the Category

ELSE

ENDIF

;Bag Ready to Washing Machine
IF (STEP = 5) THEN
	O_BagReady 		= TRUE

	IF I_OpenBag OR TestDischarger THEN
		D[914] = 6
	ENDIF
ELSE
	O_BagReady = FALSE
ENDIF

;Set LoadDropped to False
IF (STEP <> 6) THEN
	LoadDropped = FALSE
ENDIF

;Open Bag Until LoadDropped recieved and has been open for 6 seconds
TON_10ms((STEP = 6),600,MinOpen,MinOpenET) ;ET means Elapsed Time
TON_10ms((STEP = 6) AND NOT I_DischargerBagEmpty ,100,BagEmpty,BagEmptyET)

IF (STEP = 6) THEN

	;IF I_LoadDropped  OR TestDischarger THEN

		LoadDropped = TRUE
	;ENDIF

	IF (LoadDropped AND MinOpen) THEN
		;Write Report
		;------------

	ENDIF
	IF (LoadDropped AND MinOpen ) THEN
		IF (ReportUnloading[9].Cat = 0) THEN
			ReportUnloading[9].Cat = UINT(Bag[100].Cat)	;Category
			ReportUnloading[9].Cus = Bag[100].Cus		;Customer
			ReportUnloading[9].Wgt = Bag[100].Wgt		;Weight
			ReportUnloading[9].Cnt = 0					;Count
			ReportUnloading[9].Stn = 0					;Station
			ReportUnloading[9].Mcn = 9					;Machine
		ENDIF
		D[914] = 7
	ENDIF
	Alarm[14].Time			= 600
	Alarm[14].Name = almLoadNotDropped
	ELSE
	LoadDropped = FALSE
ENDIF

;Change display to empty bag
IF (STEP = 7) THEN
	IF ((NOT I_OpenBag  AND I_BagEmpty) OR TestDrop) THEN
		Bag[100].Prg 	= Std.MaxProg
		Bag[100].Cat 	= Std.MaxCats
		Bag[100].Cus 	= Std.MaxCust

		D[914] 			= 8
	ENDIF
	Alarm[14].Name = almGeneralSequence
ENDIF

;Allow steadys to go up
TON_10ms((STEP = 8),400,SteadyUp,SteadyUpET)
IF (STEP = 8) THEN
	IF SteadyUp THEN
		D[914] = 9
	ENDIF
ENDIF

;Request empty bag release
IF (STEP = 9) THEN
	Request.DCEmptyRelease[9] = TRUE
	IF Enable.DCEmptyRelease[9] THEN
		;C[32]  = 0
		D[914] = 10
	ENDIF
ENDIF

;Open buffer stop - unitl bag out
IF (STEP = 10) THEN
	O_OpenStop = TRUE
	Bag[100].Cat = 0
	Bag[100].Cus = 0
	Bag[100].Wgt = 0
	IF NOT Enable.DCEmptyRelease[9] THEN
		D[914] = 1
	ENDIF
	Alarm[14].Name = almBagNotReleased
ENDIF

;Alarms
TimerAlarm.IN 	= NOT PLS AND (Alarm[14].Name > 0)
TimerAlarm.PT 	= Alarm[14].Time
TimerAlarm FUB TON_10ms()
Alarm[14].On 	= TimerAlarm.Q
Alarm[14].ET 	= TimerAlarm.ET

;Outputs
Y[2].Y10 = O_OpenBuffer
Y[2].Y12 = O_Steadys
Y[2].Y14 = O_OpenBag
Y[2].Y11 = O_OpenStop
Y[2].Y13 = O_BagReady
END_PROGRAM
```

### Program Logical/Sequences/10ms/15_cbc1 (IEC, version 1.00.0) - * SDC2 Machine 2 CAN

#### 7_sdc2Cyclic.ab
```automation-basic
PROGRAM _CYCLIC
	(* cyclic program *)

;Sequence 7 - Discharger 2 D[907]

;-----------------------------------------
;Revision 1.00 19/12/2005 D.J. First Issue
;-----------------------------------------

DischargerEnable 		= ((D[10] > 0) AND NOT Std.HaltSys)

;I_BagAtBuffer			= X[6].X07
;I_OpenBag				= CAN[2].DropLoad OR TestDrop
;I_LoadDropped			= CAN[2].LoadDropped OR TestDropped
I_BagAtBuffer			= X[7].X05 OR TestBuffer
I_BagAtDischarger		= X[7].X06 OR TestAtDisch
I_BagEmpty			  	= TRUE

I_BagAtEmptyBuffer		= FALSE ;X[6].X13
O_EmptyBagBufferOpen	= FALSE ;Y[6].Y13

O_BagReady				= FALSE
O_OpenBuffer 			= FALSE
O_Steadys				= FALSE
O_Closer				= FALSE
O_OpenBag				= FALSE
O_OpenStop				= FALSE

;Alarm
Alarm[15].Name 			= almNoAlarm ;Clear sequence alarm name
Alarm[15].Bag 			= 10012
Alarm[15].Beacon			= TRUE
Alarm[15].Extra			= 0
Alarm[15].Time			= 3000

;Setup Sequence
STEP = D[915]
;Setup Pulse contact
PLS = (STEP <> LASTSTEP)
LASTSTEP = STEP

;Step 0 - Disabled
IF (STEP = 0) THEN
	;Disabled
ENDIF

;Check Status - Bag settled at buffer, no bag at discharger, bag at buffer on screen and no bag at discharger on the screen
TON_10ms(I_BagAtBuffer,300,SettledAtBuffer,SettledAtBufferET)
IF (STEP = 1) THEN
	IF (NOT I_BagAtDischarger  AND NOT Std.HaltSys AND DischargerEnable AND SettledAtBuffer) THEN

		D[915] = 2
	ENDIF
	IF I_BagAtDischarger THEN
		;D[907] = 2
	ENDIF

ENDIF

;Wait for bag in discharger
IF (STEP = 2) THEN
	O_OpenBuffer 	= TRUE
	IF I_BagAtDischarger THEN
		D[915] = 3
	ENDIF
	Alarm[15].Name = almNoAlarm ;almBagNotArrived
ENDIF

;Let bag settle in discharger
TON_10ms(((STEP = 3) AND I_BagAtDischarger),1000,SettledAtDischarger,SettledAtDischargerET)
IF (STEP = 3) THEN

	IF SettledAtDischarger THEN
		D[915] = 4
	ENDIF
	Alarm[15].Name = almBagNotSettled
ENDIF

;Allow steadys to move down
TON_10ms((STEP = 4),400,SteadysDown,SteadysDownET)
IF (STEP = 4) THEN
	IF SteadysDown THEN
		D[915] = 5
	ENDIF

ENDIF

;Steady cylinders on from steps 4 - 9
O_Steadys = ((STEP >= 4) AND (STEP <= 6))

;Bag opener on from step 5 - 8
O_OpenBag = ((STEP >= 5) AND (STEP <= 5))

;Close bag
TON_10ms((STEP = 5),700,CloserDown,CloserDownET)
IF (STEP = 5) THEN
	O_Closer = TRUE
	IF CloserDown THEN
		D[915] = 6
	ENDIF
ENDIF

;Allow closer to go back up
TON_10ms((STEP = 6),700,CloserUp,CloserUpET)
IF (STEP = 6) THEN
	IF CloserUp THEN
		D[915] = 7
	ENDIF
ENDIF

;Allow steadys to go up
TON_10ms((STEP = 7),400,SteadyUp,SteadyUpET)
IF (STEP = 7) THEN
	IF SteadyUp THEN
		D[915] = 8
	ENDIF
ENDIF

;Request empty bag release
IF (STEP = 8) THEN

	IF Line[30].Clear THEN
		C[30]  = 0
		D[915] = 9
	ENDIF
ENDIF

;Open buffer stop - unitl bag out
IF (STEP = 9) THEN
	O_OpenStop = TRUE

	IF Line[30].Trip THEN
		D[915] = 1
	ENDIF
	Alarm[15].Name = almBagNotReleased
ENDIF

;Alarms
TimerAlarm.IN 	= NOT PLS AND (Alarm[15].Name > 0)
TimerAlarm.PT 	= Alarm[15].Time
TimerAlarm FUB TON_10ms()
Alarm[15].On 	= TimerAlarm.Q
Alarm[15].ET 	= TimerAlarm.ET

;Outputs
Y[7].Y09 = O_OpenBuffer
Y[7].Y10 = O_Steadys
Y[7].Y11 = O_OpenBag
Y[7].Y13 = O_OpenStop
Y[7].Y12 = O_Closer
END_PROGRAM
```

### Program Logical/Sequences/10ms/16_cic1 (IEC, version 1.00.5) - *incline

#### ic.st - Implementation code
```iecst
(********************************************************************
 * COPYRIGHT --
 ********************************************************************
 * Program: ic
 * File: ic.st
 * Author: treamsbottom
 * Created: July 17, 2015
 ********************************************************************
 * Implementation of program Incline conveyor.
 ********************************************************************)
//V1.00.1 First Release
PROGRAM _INIT
//Configuration
mySeq					:= 16;		//Sequence number
myIO					:= 5; 	//Incline Conveyor IO module number
myIC					:= 1;		//Incline Conveyor Number
useRequest				:= FALSE; 	//Use the Request bit. Only use when working with x_1_point. otherwise use RequestRelease as the i_bagAtBuffer.
myBuffBag				:= 77;		//Ingoing Buffer bag number
myBag					:= 76;		//Incline bag number
myRelLine				:= 0;
myOutBag				:= 75;	//Outgoing buffer bag number

myZone 					:= 0;
//Timer Values
bufferSettleTime		:= 300;  	// Time for bag to settle at buffer in.
moveUpInclineTime		:= 4;//>>IN SECONDS<< // Time to move bag up incline after closing stop.//Min of 4 to shut buffer stop....

alarm						ACCESS ADR(Alarm[mySeq]);
bag							ACCESS ADR(Bag[myBag]);
bag_buff					ACCESS ADR(Bag[myBuffBag]);
bag_out						ACCESS ADR(Bag[myOutBag]);
line_release				ACCESS ADR(Line[myRelLine]);
END_PROGRAM

PROGRAM _CYCLIC
//Inputs
i_paddleInPosition		:= X[myIO].X09;
i_bagAtBuffer			:= X[myIO].X08;
i_bagInIncline			:= X[myIO].X10;
i_BagReleased			:= FALSE;//X[myIO].X05;  //<--- Bag release trip- only to be used in special cases. Take when using tracked bags, as the next sequence will need to copy data into a transit position

i_bagAtBufferOut 		:= FALSE; // Any Single bag buffer out IO.
i_bufferOutOpen			:= FALSE;

//End of inputs.

o_openBuffer			:= FALSE;
o_runMotor				:= FALSE;

Request.IC[myIC] 		:= FALSE;
RequestRel.IC[myIC] 	:= FALSE;

IF (myBag = 0) THEN
	alarm.Bag	:= mySeq + 10000;
ELSE
	alarm.Bag	:= myBag;
END_IF;

alarm.Name 		:= 0;
alarm.Beacon		:= TRUE;
alarm.Extra		:= 0;
alarm.Time		:= 3000;

//Setup Sequence
step := D[900 + mySeq];
//Setup Pulse contact
pls := (step <> laststep);
laststep := step;

//Sequence
IF (step = 0) THEN
	//Disabled
END_IF;

//Run Incline until paddle in position
IF (step = 1) THEN
	o_runMotor := NOT i_paddleInPosition;
	IF i_paddleInPosition THEN
		D[900 + mySeq] := 2;
		Count[mySeq] := Count[mySeq] + 1;
	END_IF;
	IF NOT Std.HaltSysZone[myZone] THEN
		alarm.Name := ALM_SWITCH_FAULT;
	END_IF;
END_IF;

//Wait for at buffer
ton_10ms_SettledBuffer(IN:= i_bagAtBuffer, PT:= bufferSettleTime);
IF (step = 2) THEN
	IF NOT i_bagInIncline THEN
		IF useRequest THEN
			D[900 + mySeq] := 3;
		ELSE
			IF ton_10ms_SettledBuffer.Q THEN
				IF (myBuffBag > 0) THEN
					IF (bag_buff.Cat > 0) AND (bag.Cat = 0) THEN
						D[900 + mySeq] := 3;
					ELSIF (bag_buff.Cat = 0) THEN
						alarm.Name := ALM_BAG_DATA_ERROR;
						alarm.Bag := myBuffBag;
					ELSE
						alarm.Name := ALM_BAG_DATA_ERROR;
					END_IF;
				ELSE
					D[900 + mySeq] := 3;
				END_IF;
			ELSIF (myBuffBag > 0) AND (bag_buff.Cat > 0) THEN
				alarm.Name := ALM_BAG_NOT_SETTLED;
			END_IF;
		END_IF;
	ELSE
		alarm.Name := ALM_SWITCH_FAULT;
	END_IF;
END_IF;

//Open Buffer stop
IF (step = 3) THEN
	releaseValid := ((myBag = 0) OR ((bag.Cat = 0) AND (bag_buff.Cat > 0)));
	o_openBuffer	   := releaseValid AND NOT useRequest;
	Request.IC[myIC]  := releaseValid AND useRequest;
	IF i_bagInIncline AND releaseValid THEN
		IF (myBag > 0) THEN
			bag := bag_buff; //Clear empty buffer bag data if used
			bag_buff := Bag[0];
		END_IF;
		D[900 + mySeq] := 4;
	ELSIF (myBag > 0) THEN
		IF (bag.Cat > 0) THEN
			alarm.Name := ALM_BAG_DATA_ERROR;
			alarm.Time := 0;
		ELSIF (bag_buff.Cat = 0) THEN
			alarm.Name := ALM_BAG_DATA_ERROR;
			alarm.Bag := myBuffBag;
			alarm.Time := 0;
		ELSE
			alarm.Name  := ALM_BAG_NOT_ARRIVED;
		END_IF;
	ELSE
		alarm.Name  := ALM_BAG_NOT_ARRIVED;
	END_IF;
END_IF;

ton_10ms_SettledIncline(IN:= (step = 4), PT:= 300);
IF (step = 4) THEN
	o_openBuffer := NOT useRequest;
	IF ton_10ms_SettledIncline.Q THEN
		D[900 + mySeq] := 5;
	END_IF;
END_IF;

//Move Bag up incline
ctu_moveUpIncline(CU:=(step = 5) AND NOT Std.HaltSysZone[myZone] AND Std.Clock1s, RESET := (step <> 5), PV := moveUpInclineTime);
IF (step = 5) THEN
	o_openBuffer 	:= (ctu_moveUpIncline.CV <= 4) AND NOT useRequest;//Close buffer stop after 3 seconds running..
	o_runMotor 		:= TRUE;
	IF ctu_moveUpIncline.Q THEN
		D[900 + mySeq] := 6;
	ELSIF NOT Std.HaltSysZone[myZone] THEN
		alarm.Name := ALM_SWITCH_FAULT;
	END_IF;

END_IF;

//Check for line space.
IF (step = 6) THEN
	CDC4Release := (NOT i_bagAtBufferOut AND NOT i_bufferOutOpen AND NOT i_BagReleased AND ((myBag = 0) OR ((bag.Cat > 0))));
	releaseValid := NOT i_bagAtBufferOut; //AND NOT i_bufferOutOpen AND NOT i_BagReleased AND  (bag.Cat > 0);
	IF (myRelLine > 0) THEN
		IF (line_release.Clear AND releaseValid) THEN
			C[myRelLine] := 0;
			D[900 + mySeq] := 7;
		END_IF;
		IF (line_release.Clear AND i_bagAtBufferOut) THEN
			alarm.Name := ALM_SWITCH_FAULT;
		ELSIF (myBag > 0) AND (bag.Cat = 0) THEN
			alarm.Name := ALM_BAG_DATA_ERROR;
			alarm.Time := 0;
		ELSIF line_release.Clear AND (myOutBag > 0) AND (bag_out.Cat > 0) THEN
			alarm.Name := ALM_BAG_DATA_ERROR;
			alarm.Bag := myOutBag;
			alarm.Time := 0;
		END_IF;
	ELSE
		RequestRel.IC[myIC] := (releaseValid OR CDC4Release);
		IF EnableRel.IC[myIC] AND releaseValid THEN

			D[900 + mySeq] := 7;
		ELSIF (myBag > 0) AND (bag.Cat = 0) THEN
			alarm.Name := ALM_BAG_DATA_ERROR;
			alarm.Time := 0;
		ELSIF (myOutBag > 0) AND (bag_out.Cat > 0) THEN
	//	;	alarm.Name := ALM_BAG_DATA_ERROR;
	//	;	alarm.Bag := myOutBag;
		//	alarm.Time := 0;
		END_IF;
	END_IF;
	IF i_BagReleased THEN
		alarm.Name := ALM_SWITCH_FAULT;
		alarm.Time := 0;
	END_IF;
	releaseValid := 0; //Clear this as we are using it as a latch in line 7
END_IF;

//Run motor to release bag.
IF (step = 7) THEN
	IF (NOT i_bagAtBufferOut AND NOT i_bufferOutOpen AND ((myBag = 0) OR ((bag.Cat > 0) AND (bag_out.Cat = 0)))) THEN
		releaseValid := 1;
	END_IF;
	o_runMotor := releaseValid AND NOT Std.HaltSysZone[myZone];
	IF o_runMotor THEN
		alarm.Time := 1000;
		alarm.Name := ALM_BAG_NOT_RELEASED;
	END_IF
	IF releaseValid THEN
		IF (myBag = 0) THEN
			IF (myRelLine > 0) THEN
				IF line_release.Trip THEN
					D[900 + mySeq] := 1;
				END_IF;
			ELSE
				IF NOT EnableRel.IC[myIC] OR i_BagReleased THEN
					D[900 + mySeq] := 1;
				END_IF;
			END_IF;
			IF NOT Std.HaltSysZone[myZone] THEN
				alarm.Name := ALM_BAG_NOT_RELEASED;
			END_IF;
		ELSE//Use tracking
			IF (myRelLine > 0) THEN
				IF line_release.Trip THEN
					bag_out := bag;
					bag := Bag[0];
					D[900 + mySeq] := 1;
				END_IF;
			ELSE
				IF (i_BagReleased OR NOT EnableRel.IC[myIC]) AND (bag.Cat = 0)  THEN // Make sure data is copied out by enabling sequence.
					D[900 + mySeq] := 1;
				ELSIF NOT EnableRel.IC[myIC] AND (bag.Cat > 0) THEN
					alarm.Name := ALM_BAG_DATA_ERROR;
				END_IF;
			END_IF;
		END_IF;
	ELSIF i_bagAtBufferOut OR i_bufferOutOpen THEN
			alarm.Name := ALM_SWITCH_FAULT;
			alarm.Time := 0;
	ELSIF (myBag > 0) THEN
		IF (bag.Cat = 0) THEN
			alarm.Name := ALM_BAG_DATA_ERROR;
			alarm.Time := 0;
		ELSIF (bag_out.Cat > 0) THEN
			alarm.Name := ALM_BAG_DATA_ERROR;
			alarm.Bag := myOutBag;
			alarm.Time := 0;
		END_IF;
	END_IF;
END_IF;

//-----------------------------------
//PLC Outputs - adjust TO suit system
//-----------------------------------

Y[11].Y04	:= o_runMotor;
Y[4].Y13 := o_openBuffer;

//Alarms
timerAlarm(IN := NOT pls AND (alarm.Name > 0),PT:= alarm.Time);

alarm.On 	:= timerAlarm.Q;
alarm.ET 	:= timerAlarm.ET;;

END_PROGRAM
```

#### ic.var - Local variables
```iecst
(********************************************************************
 * COPYRIGHT --
 ********************************************************************
 * Program: ic
 * File: ic.var
 * Author: treamsbottom
 * Created: July 17, 2015
 ********************************************************************
 * Local variables of program ic
 ********************************************************************)
VAR
	mySeq : UINT;
	myIO : UINT;
	myIC : UINT;
	useRequest : BOOL;
	bufferSettleTime : UDINT;
	myBuffBag : UINT;
	myBag : UINT;
	myRelLine : UINT;
	myOutBag : UINT;
	myZone : UINT;
	i_paddleInPosition : BOOL;
	i_bagAtBuffer : BOOL;
	i_bagAtBufferOut : BOOL;
	i_bufferOutOpen : BOOL;
	o_openBuffer : BOOL;
	o_runMotor : BOOL;
	step : UINT;
	pls : BOOL;
	ton_10ms_SettledBuffer : TON_10ms;
	timerAlarm : TON_10ms;
END_VAR
VAR RETAIN
	laststep : UINT;
END_VAR
VAR
	i_bagInIncline : BOOL;
	moveUpInclineTime : UINT;
	releaseValid : BOOL;
	ton_10ms_SettledIncline : TON_10ms;
	ctu_moveUpIncline : CTU;
	i_BagReleased : BOOL;
	alarm : REFERENCE TO Alm;
	bag : REFERENCE TO Bag_typ;
	bag_buff : REFERENCE TO Bag_typ;
	bag_out : REFERENCE TO Bag_typ;
	line_release : REFERENCE TO Line_Typ;
	CDC4Release : BOOL;
END_VAR
```

### Program Logical/Sequences/10ms/17_cic2 (IEC) - *incline

#### ic.st
```iecst
(********************************************************************
 * COPYRIGHT --
 ********************************************************************
 * Program: ic
 * File: ic.st
 * Author: treamsbottom
 * Created: July 17, 2015
 ********************************************************************
 * Implementation of program Incline conveyor.
 ********************************************************************)
//V1.00.1 First Release
PROGRAM _INIT
//Configuration
mySeq					:= 17;		//Sequence number
myIO					:= 171; 	//Incline Conveyor IO module number
myIC					:= 2;		//Incline Conveyor Number
useRequest				:= FALSE; 	//Use the Request bit. Only use when working with x_1_point. otherwise use RequestRelease as the i_bagAtBuffer.
myBuffBag				:= 146;		//Ingoing Buffer bag number
myBag					:= 154;		//Incline bag number
myRelLine				:= 0;
myOutBag				:= Line[myRelLine].LastBag;	//Outgoing buffer bag number

myZone 					:= 0;
//Timer Values
bufferSettleTime		:= 300;  	// Time for bag to settle at buffer in.
moveUpInclineTime		:= 10;//>>IN SECONDS<< // Time to move bag up incline after closing stop.//Min of 4 to shut buffer stop....

alarm						ACCESS ADR(Alarm[mySeq]);
bag							ACCESS ADR(Bag[myBag]);
bag_buff					ACCESS ADR(Bag[myBuffBag]);
bag_out						ACCESS ADR(Bag[myOutBag]);
line_release				ACCESS ADR(Line[myRelLine]);
END_PROGRAM

PROGRAM _CYCLIC
//Inputs
i_paddleInPosition		:= X[5].X12;
i_bagAtBuffer			:= X[5].X11;
i_bagInIncline			:= X[5].X13;
i_BagReleased			:= FALSE;//X[myIO].X05;  //<--- Bag release trip- only to be used in special cases. Take when using tracked bags, as the next sequence will need to copy data into a transit position

i_bagAtBufferOut 		:= FALSE; // Any Single bag buffer out IO.
i_bufferOutOpen			:= FALSE;

//End of inputs.

o_openBuffer			:= FALSE;
o_runMotor				:= FALSE;

Request.IC[myIC] 		:= FALSE;
RequestRel.IC[myIC] 	:= FALSE;

IF (myBag = 0) THEN
	alarm.Bag	:= mySeq + 10000;
ELSE
	alarm.Bag	:= myBag;
END_IF;

alarm.Name 		:= 0;
alarm.Beacon		:= TRUE;
alarm.Extra		:= 0;
alarm.Time		:= 3000;

//Setup Sequence
step := D[900 + mySeq];
//Setup Pulse contact
pls := (step <> laststep);
laststep := step;

//Sequence
IF (step = 0) THEN
	//Disabled
END_IF;

//Run Incline until paddle in position
IF (step = 1) THEN
	o_runMotor := NOT i_paddleInPosition;
	IF i_paddleInPosition THEN
		D[900 + mySeq] := 2;
		Count[mySeq] := Count[mySeq] + 1;
	END_IF;
	IF NOT Std.HaltSysZone[myZone] THEN
		alarm.Name := ALM_SWITCH_FAULT;
	END_IF;
END_IF;

//Wait for at buffer
ton_10ms_SettledBuffer(IN:= i_bagAtBuffer, PT:= bufferSettleTime);
IF (step = 2) THEN
	IF NOT i_bagInIncline THEN
		IF useRequest THEN
			D[900 + mySeq] := 3;
		ELSE
			IF ton_10ms_SettledBuffer.Q THEN
				IF (myBuffBag > 0) THEN
					IF (bag_buff.Cat > 0) AND (bag.Cat = 0) THEN
						D[900 + mySeq] := 3;
					ELSIF (bag_buff.Cat = 0) THEN
						alarm.Name := ALM_BAG_DATA_ERROR;
						alarm.Bag := myBuffBag;
					ELSE
						alarm.Name := ALM_BAG_DATA_ERROR;
					END_IF;
				ELSE
					D[900 + mySeq] := 3;
				END_IF;
			ELSIF (myBuffBag > 0) AND (bag_buff.Cat > 0) THEN
				alarm.Name := ALM_BAG_NOT_SETTLED;
			END_IF;
		END_IF;
	ELSE
		alarm.Name := ALM_SWITCH_FAULT;
	END_IF;
END_IF;

//Open Buffer stop
IF (step = 3) THEN
	releaseValid := ((myBag = 0) OR ((bag.Cat = 0) AND (bag_buff.Cat > 0)));
	o_openBuffer	   := releaseValid AND NOT useRequest;
	Request.IC[myIC]  := releaseValid AND useRequest;
	IF i_bagInIncline AND releaseValid THEN
		IF (myBag > 0) THEN
			bag := bag_buff; //Clear empty buffer bag data if used
			bag_buff := Bag[0];
		END_IF;
		D[900 + mySeq] := 4;
	ELSIF (myBag > 0) THEN
		IF (bag.Cat > 0) THEN
			alarm.Name := ALM_BAG_DATA_ERROR;
			alarm.Time := 0;
		ELSIF (bag_buff.Cat = 0) THEN
			alarm.Name := ALM_BAG_DATA_ERROR;
			alarm.Bag := myBuffBag;
			alarm.Time := 0;
		ELSE
			alarm.Name  := ALM_BAG_NOT_ARRIVED;
		END_IF;
	ELSE
		alarm.Name  := ALM_BAG_NOT_ARRIVED;
	END_IF;
END_IF;

ton_10ms_SettledIncline(IN:= (step = 4), PT:= 300);
IF (step = 4) THEN
	o_openBuffer := NOT useRequest;
	IF ton_10ms_SettledIncline.Q THEN
		D[900 + mySeq] := 5;
	END_IF;
END_IF;

//Move Bag up incline
ctu_moveUpIncline(CU:=(step = 5) AND NOT Std.HaltSysZone[myZone] AND Std.Clock1s, RESET := (step <> 5), PV := moveUpInclineTime);
IF (step = 5) THEN
	o_openBuffer 	:= (ctu_moveUpIncline.CV <= 4) AND NOT useRequest;//Close buffer stop after 3 seconds running..
	o_runMotor 		:= TRUE;
	IF ctu_moveUpIncline.Q THEN
		D[900 + mySeq] := 6;
	ELSIF NOT Std.HaltSysZone[myZone] THEN
		alarm.Name := ALM_SWITCH_FAULT;
	END_IF;

END_IF;

//Check for line space.
IF (step = 6) THEN
	releaseValid := TRUE;//(NOT i_bagAtBufferOut AND NOT i_bufferOutOpen AND NOT i_BagReleased AND ((myBag = 0) OR ((bag.Cat > 0) AND (bag_out.Cat = 0))));
	IF (myRelLine > 0) THEN
		IF (line_release.Clear AND releaseValid) THEN
			C[myRelLine] := 0;
			D[900 + mySeq] := 7;
		END_IF;
		IF (line_release.Clear AND i_bagAtBufferOut) THEN
			alarm.Name := ALM_SWITCH_FAULT;
		ELSIF (myBag > 0) AND (bag.Cat = 0) THEN
			alarm.Name := ALM_BAG_DATA_ERROR;
			alarm.Time := 0;
		ELSIF line_release.Clear AND (myOutBag > 0) AND (bag_out.Cat > 0) THEN
			alarm.Name := ALM_BAG_DATA_ERROR;
			alarm.Bag := myOutBag;
			alarm.Time := 0;
		END_IF;
	ELSE
		RequestRel.IC[myIC] := releaseValid;
		IF EnableRel.IC[myIC] AND releaseValid THEN

			D[900 + mySeq] := 7;
		ELSIF (myBag > 0) AND (bag.Cat = 0) THEN
			alarm.Name := ALM_BAG_DATA_ERROR;
			alarm.Time := 0;
		ELSIF (myOutBag > 0) AND (bag_out.Cat > 0) THEN
			alarm.Name := ALM_BAG_DATA_ERROR;
			alarm.Bag := myOutBag;
			alarm.Time := 0;
		END_IF;
	END_IF;
	IF i_BagReleased THEN
		alarm.Name := ALM_SWITCH_FAULT;
		alarm.Time := 0;
	END_IF;
	releaseValid := 0; //Clear this as we are using it as a latch in line 7
END_IF;

//Run motor to release bag.
IF (step = 7) THEN
	IF (NOT i_bagAtBufferOut AND NOT i_bufferOutOpen AND ((myBag = 0) OR ((bag.Cat > 0) AND (bag_out.Cat = 0)))) THEN
		releaseValid := 1;
	END_IF;
	o_runMotor := releaseValid AND NOT Std.HaltSysZone[myZone];
	IF releaseValid THEN
		IF (myBag = 0) THEN
			IF (myRelLine > 0) THEN
				IF line_release.Trip THEN
					D[900 + mySeq] := 1;
				END_IF;
			ELSE
				IF NOT EnableRel.IC[myIC] OR i_BagReleased THEN
					D[900 + mySeq] := 1;
				END_IF;
			END_IF;
			IF NOT Std.HaltSysZone[myZone] THEN
				alarm.Name := ALM_BAG_NOT_RELEASED;
			END_IF;
		ELSE//Use tracking
			IF (myRelLine > 0) THEN
				IF line_release.Trip THEN
					bag_out := bag;
					bag := Bag[0];
					D[900 + mySeq] := 1;
				END_IF;
			ELSE
				IF (i_BagReleased OR NOT EnableRel.IC[myIC]) AND (bag.Cat = 0)  THEN // Make sure data is copied out by enabling sequence.
					D[900 + mySeq] := 1;
				ELSIF NOT EnableRel.IC[myIC] AND (bag.Cat > 0) THEN
					alarm.Name := ALM_BAG_DATA_ERROR;
				END_IF;
			END_IF;
		END_IF;
	ELSIF i_bagAtBufferOut OR i_bufferOutOpen THEN
			alarm.Name := ALM_SWITCH_FAULT;
			alarm.Time := 0;
	ELSIF (myBag > 0) THEN
		IF (bag.Cat = 0) THEN
			alarm.Name := ALM_BAG_DATA_ERROR;
			alarm.Time := 0;
		ELSIF (bag_out.Cat > 0) THEN
			alarm.Name := ALM_BAG_DATA_ERROR;
			alarm.Bag := myOutBag;
			alarm.Time := 0;
		END_IF;
	END_IF;
END_IF;

//-----------------------------------
//PLC Outputs - adjust TO suit system
//-----------------------------------

Y[11].Y05	:= o_runMotor;
Y[4].Y14 := o_openBuffer;

//Alarms
timerAlarm(IN := NOT pls AND (alarm.Name > 0),PT:= alarm.Time);

alarm.On 	:= timerAlarm.Q;
alarm.ET 	:= timerAlarm.ET;;

END_PROGRAM
```

### Program Logical/Sequences/10ms/18_cic3 (IEC) - *incline

#### ic.st
```iecst
(********************************************************************
 * COPYRIGHT --
 ********************************************************************
 * Program: ic
 * File: ic.st
 * Author: treamsbottom
 * Created: July 17, 2015
 ********************************************************************
 * Implementation of program Incline conveyor.
 ********************************************************************)
//V1.00.1 First Release
PROGRAM _INIT
//Configuration
mySeq					:= 18;		//Sequence number
myIO					:= 8; 	//Incline Conveyor IO module number
myIC					:= 3;		//Incline Conveyor Number
useRequest				:= FALSE; 	//Use the Request bit. Only use when working with x_1_point. otherwise use RequestRelease as the i_bagAtBuffer.
myBuffBag				:= 0;		//Ingoing Buffer bag number
myBag					:= 0;		//Incline bag number
myRelLine				:= 10;
myOutBag				:= Line[myRelLine].LastBag;	//Outgoing buffer bag number

myZone 					:= 0;
//Timer Values
bufferSettleTime		:= 300;  	// Time for bag to settle at buffer in.
moveUpInclineTime		:= 4;//>>IN SECONDS<< // Time to move bag up incline after closing stop.//Min of 4 to shut buffer stop....

alarm						ACCESS ADR(Alarm[mySeq]);
bag							ACCESS ADR(Bag[myBag]);
bag_buff					ACCESS ADR(Bag[myBuffBag]);
bag_out						ACCESS ADR(Bag[myOutBag]);
line_release				ACCESS ADR(Line[myRelLine]);
END_PROGRAM

PROGRAM _CYCLIC
//Inputs
i_paddleInPosition		:= X[myIO].X09;
i_bagAtBuffer			:= X[myIO].X08;
i_bagInIncline			:= X[myIO].X10;
i_BagReleased			:= FALSE;//X[myIO].X05;  //<--- Bag release trip- only to be used in special cases. Take when using tracked bags, as the next sequence will need to copy data into a transit position

i_bagAtBufferOut 		:= FALSE; // Any Single bag buffer out IO.
i_bufferOutOpen			:= FALSE;

//End of inputs.

o_openBuffer			:= FALSE;
o_runMotor				:= FALSE;

Request.IC[myIC] 		:= FALSE;
RequestRel.IC[myIC] 	:= FALSE;

IF (myBag = 0) THEN
	alarm.Bag	:= mySeq + 10000;
ELSE
	alarm.Bag	:= myBag;
END_IF;

alarm.Name 		:= 0;
alarm.Bag	:= 10011;
alarm.Beacon		:= TRUE;
alarm.Extra		:= 0;
alarm.Time		:= 3000;

//Setup Sequence
step := D[900 + mySeq];
//Setup Pulse contact
pls := (step <> laststep);
laststep := step;

//Sequence
IF (step = 0) THEN
	//Disabled
END_IF;

//Run Incline until paddle in position
IF (step = 1) THEN
	o_runMotor := NOT i_paddleInPosition;
	IF i_paddleInPosition THEN
		D[900 + mySeq] := 2;
		Count[mySeq] := Count[mySeq] + 1;
	END_IF;
	IF NOT Std.HaltSysZone[myZone] THEN
		alarm.Name := ALM_SWITCH_FAULT;
	END_IF;
END_IF;

//Wait for at buffer
ton_10ms_SettledBuffer(IN:= i_bagAtBuffer, PT:= bufferSettleTime);
IF (step = 2) THEN
	IF NOT i_bagInIncline THEN
		IF useRequest THEN
			D[900 + mySeq] := 3;
		ELSE
			IF ton_10ms_SettledBuffer.Q THEN
				IF (myBuffBag > 0) THEN
					IF (bag_buff.Cat > 0) AND (bag.Cat = 0) THEN
						D[900 + mySeq] := 3;
					ELSIF (bag_buff.Cat = 0) THEN
						alarm.Name := ALM_BAG_DATA_ERROR;
						alarm.Bag := myBuffBag;
					ELSE
						alarm.Name := ALM_BAG_DATA_ERROR;
					END_IF;
				ELSE
					D[900 + mySeq] := 3;
				END_IF;
			ELSIF (myBuffBag > 0) AND (bag_buff.Cat > 0) THEN
				alarm.Name := ALM_BAG_NOT_SETTLED;
			END_IF;
		END_IF;
	ELSE
		alarm.Name := ALM_SWITCH_FAULT;
	END_IF;
END_IF;

//Open Buffer stop
IF (step = 3) THEN
	releaseValid := ((myBag = 0) OR ((bag.Cat = 0) AND (bag_buff.Cat > 0)));
	o_openBuffer	   := releaseValid AND NOT useRequest;
	Request.IC[myIC]  := releaseValid AND useRequest;
	IF i_bagInIncline AND releaseValid THEN
		IF (myBag > 0) THEN
			bag := bag_buff; //Clear empty buffer bag data if used
			bag_buff := Bag[0];
		END_IF;
		D[900 + mySeq] := 4;
	ELSIF (myBag > 0) THEN
		IF (bag.Cat > 0) THEN
			alarm.Name := ALM_BAG_DATA_ERROR;
			alarm.Time := 0;
		ELSIF (bag_buff.Cat = 0) THEN
			alarm.Name := ALM_BAG_DATA_ERROR;
			alarm.Bag := myBuffBag;
			alarm.Time := 0;
		ELSE
			alarm.Name  := ALM_BAG_NOT_ARRIVED;
		END_IF;
	ELSE
		alarm.Name  := ALM_BAG_NOT_ARRIVED;
	END_IF;
END_IF;

ton_10ms_SettledIncline(IN:= (step = 4), PT:= 300);
IF (step = 4) THEN
	o_openBuffer := NOT useRequest;
	IF ton_10ms_SettledIncline.Q THEN
		D[900 + mySeq] := 5;
	END_IF;
END_IF;

//Move Bag up incline
ctu_moveUpIncline(CU:=(step = 5) AND NOT Std.HaltSysZone[myZone] AND Std.Clock1s, RESET := (step <> 5), PV := moveUpInclineTime);
IF (step = 5) THEN
	o_openBuffer 	:= (ctu_moveUpIncline.CV <= 4) AND NOT useRequest;//Close buffer stop after 3 seconds running..
	o_runMotor 		:= TRUE;
	IF ctu_moveUpIncline.Q THEN
		D[900 + mySeq] := 6;
	ELSIF NOT Std.HaltSysZone[myZone] THEN
		alarm.Name := ALM_SWITCH_FAULT;
	END_IF;

END_IF;

//Check for line space.
IF (step = 6) THEN
	releaseValid := (NOT i_bagAtBufferOut AND NOT i_bufferOutOpen AND NOT i_BagReleased AND ((myBag = 0) OR ((bag.Cat > 0) AND (bag_out.Cat = 0))));
	IF (myRelLine > 0) THEN
		IF (line_release.Clear AND releaseValid) THEN
			C[myRelLine] := 0;
			D[900 + mySeq] := 7;
		END_IF;
		IF (line_release.Clear AND i_bagAtBufferOut) THEN
			alarm.Name := ALM_SWITCH_FAULT;
		ELSIF (myBag > 0) AND (bag.Cat = 0) THEN
			alarm.Name := ALM_BAG_DATA_ERROR;
			alarm.Time := 0;
		ELSIF line_release.Clear AND (myOutBag > 0) AND (bag_out.Cat > 0) THEN
			alarm.Name := ALM_BAG_DATA_ERROR;
			alarm.Bag := myOutBag;
			alarm.Time := 0;
		END_IF;
	ELSE
		RequestRel.IC[myIC] := releaseValid;
		IF EnableRel.IC[myIC] AND releaseValid THEN

			D[900 + mySeq] := 7;
		ELSIF (myBag > 0) AND (bag.Cat = 0) THEN
			alarm.Name := ALM_BAG_DATA_ERROR;
			alarm.Time := 0;
		ELSIF (myOutBag > 0) AND (bag_out.Cat > 0) THEN
			alarm.Name := ALM_BAG_DATA_ERROR;
			alarm.Bag := myOutBag;
			alarm.Time := 0;
		END_IF;
	END_IF;
	IF i_BagReleased THEN
		alarm.Name := ALM_SWITCH_FAULT;
		alarm.Time := 0;
	END_IF;
	releaseValid := 0; //Clear this as we are using it as a latch in line 7
END_IF;

//Run motor to release bag.
IF (step = 7) THEN
	IF (NOT i_bagAtBufferOut AND NOT i_bufferOutOpen AND ((myBag = 0) OR ((bag.Cat > 0) AND (bag_out.Cat = 0)))) THEN
		releaseValid := 1;
	END_IF;
	o_runMotor := releaseValid AND NOT Std.HaltSysZone[myZone];
	IF releaseValid THEN
		IF (myBag = 0) THEN
			IF (myRelLine > 0) THEN
				IF line_release.Trip THEN
					D[900 + mySeq] := 1;
				END_IF;
			ELSE
				IF NOT EnableRel.IC[myIC] OR i_BagReleased THEN
					D[900 + mySeq] := 1;
				END_IF;
			END_IF;
			IF NOT Std.HaltSysZone[myZone] THEN
				alarm.Name := ALM_BAG_NOT_RELEASED;
			END_IF;
		ELSE//Use tracking
			IF (myRelLine > 0) THEN
				IF line_release.Trip THEN
					bag_out := bag;
					bag := Bag[0];
					D[900 + mySeq] := 1;
				END_IF;
			ELSE
				IF (i_BagReleased OR NOT EnableRel.IC[myIC]) AND (bag.Cat = 0)  THEN // Make sure data is copied out by enabling sequence.
					D[900 + mySeq] := 1;
				ELSIF NOT EnableRel.IC[myIC] AND (bag.Cat > 0) THEN
					alarm.Name := ALM_BAG_DATA_ERROR;
				END_IF;
			END_IF;
		END_IF;
	ELSIF i_bagAtBufferOut OR i_bufferOutOpen THEN
			alarm.Name := ALM_SWITCH_FAULT;
			alarm.Time := 0;
	ELSIF (myBag > 0) THEN
		IF (bag.Cat = 0) THEN
			alarm.Name := ALM_BAG_DATA_ERROR;
			alarm.Time := 0;
		ELSIF (bag_out.Cat > 0) THEN
			alarm.Name := ALM_BAG_DATA_ERROR;
			alarm.Bag := myOutBag;
			alarm.Time := 0;
		END_IF;
	END_IF;
END_IF;

//-----------------------------------
//PLC Outputs - adjust TO suit system
//-----------------------------------

Y[11].Y06	:= o_runMotor;
Y[4].Y15 := o_openBuffer;

//Alarms
timerAlarm(IN := NOT pls AND (alarm.Name > 0),PT:= alarm.Time);

alarm.On 	:= timerAlarm.Q;
alarm.ET 	:= timerAlarm.ET;;

END_PROGRAM
```

### Program Logical/Sequences/10ms/19_cic4 (IEC) - *incline

#### ic.st
```iecst
(********************************************************************
 * COPYRIGHT --
 ********************************************************************
 * Program: ic
 * File: ic.st
 * Author: treamsbottom
 * Created: July 17, 2015
 ********************************************************************
 * Implementation of program Incline conveyor.
 ********************************************************************)
//V1.00.1 First Release
PROGRAM _INIT
//Configuration
mySeq					:= 19;		//Sequence number
myIO					:= 9; 	//Incline Conveyor IO module number
myIC					:= 4;		//Incline Conveyor Number
useRequest				:= FALSE; 	//Use the Request bit. Only use when working with x_1_point. otherwise use RequestRelease as the i_bagAtBuffer.
myBuffBag				:= 123;		//Ingoing Buffer bag number
myBag					:= 135;		//Incline bag number
myRelLine				:= 20;
myOutBag				:= 144;	//Outgoing buffer bag number

myZone 					:= 0;
//Timer Values
bufferSettleTime		:= 300;  	// Time for bag to settle at buffer in.
moveUpInclineTime		:= 4;//>>IN SECONDS<< // Time to move bag up incline after closing stop.//Min of 4 to shut buffer stop....

alarm						ACCESS ADR(Alarm[mySeq]);
bag							ACCESS ADR(Bag[myBag]);
bag_buff					ACCESS ADR(Bag[myBuffBag]);
bag_out						ACCESS ADR(Bag[myOutBag]);
line_release				ACCESS ADR(Line[myRelLine]);
END_PROGRAM

PROGRAM _CYCLIC
//Inputs
i_paddleInPosition		:= X[myIO].X09;
i_bagAtBuffer			:= X[myIO].X10;
i_bagInIncline			:= X[myIO].X11;
i_BagReleased			:= FALSE;//X[myIO].X05;  //<--- Bag release trip- only to be used in special cases. Take when using tracked bags, as the next sequence will need to copy data into a transit position

i_bagAtBufferOut 		:= FALSE; // Any Single bag buffer out IO.
i_bufferOutOpen			:= FALSE;

//End of inputs.

o_openBuffer			:= FALSE;
o_runMotor				:= FALSE;

Request.IC[myIC] 		:= FALSE;
RequestRel.IC[myIC] 	:= FALSE;

IF (myBag = 0) THEN
	alarm.Bag	:= mySeq + 10000;
ELSE
	alarm.Bag	:= myBag;
END_IF;

alarm.Name 		:= 0;
alarm.Beacon		:= TRUE;
alarm.Extra		:= 0;
alarm.Time		:= 3000;

//Setup Sequence
step := D[900 + mySeq];
//Setup Pulse contact
pls := (step <> laststep);
laststep := step;

//Sequence
IF (step = 0) THEN
	//Disabled
END_IF;

//Run Incline until paddle in position
IF (step = 1) THEN
	o_runMotor := NOT i_paddleInPosition;
	IF i_paddleInPosition THEN
		D[900 + mySeq] := 2;
		Count[mySeq] := Count[mySeq] + 1;
	END_IF;
	IF NOT Std.HaltSysZone[myZone] THEN
		alarm.Name := ALM_SWITCH_FAULT;
	END_IF;
END_IF;

//Wait for at buffer
ton_10ms_SettledBuffer(IN:= i_bagAtBuffer, PT:= bufferSettleTime);
IF (step = 2) THEN
	IF NOT i_bagInIncline THEN
		IF useRequest THEN
			D[900 + mySeq] := 3;
		ELSE
			IF ton_10ms_SettledBuffer.Q THEN
				IF (myBuffBag > 0) THEN
					IF (bag_buff.Cat > 0) AND (bag.Cat = 0) THEN
						D[900 + mySeq] := 3;
					ELSIF (bag_buff.Cat = 0) THEN
						alarm.Name := ALM_BAG_DATA_ERROR;
						alarm.Bag := myBuffBag;
					ELSE
						alarm.Name := ALM_BAG_DATA_ERROR;
					END_IF;
				ELSE
					D[900 + mySeq] := 3;
				END_IF;
			ELSIF (myBuffBag > 0) AND (bag_buff.Cat > 0) THEN
				alarm.Name := ALM_BAG_NOT_SETTLED;
			END_IF;
		END_IF;
	ELSE
		alarm.Name := ALM_SWITCH_FAULT;
	END_IF;
END_IF;

//Open Buffer stop
IF (step = 3) THEN
	releaseValid := ((myBag = 0) OR ((bag.Cat = 0) AND (bag_buff.Cat > 0)));
	o_openBuffer	   := releaseValid AND NOT useRequest;
	Request.IC[myIC]  := releaseValid AND useRequest;
	IF i_bagInIncline AND releaseValid THEN
		IF (myBag > 0) THEN
			bag := bag_buff; //Clear empty buffer bag data if used
			bag_buff := Bag[0];
		END_IF;
		D[900 + mySeq] := 4;
	ELSIF (myBag > 0) THEN
		IF (bag.Cat > 0) THEN
			alarm.Name := ALM_BAG_DATA_ERROR;
			alarm.Time := 0;
		ELSIF (bag_buff.Cat = 0) THEN
			alarm.Name := ALM_BAG_DATA_ERROR;
			alarm.Bag := myBuffBag;
			alarm.Time := 0;
		ELSE
			alarm.Name  := ALM_BAG_NOT_ARRIVED;
		END_IF;
	ELSE
		alarm.Name  := ALM_BAG_NOT_ARRIVED;
	END_IF;
END_IF;

ton_10ms_SettledIncline(IN:= (step = 4), PT:= 300);
IF (step = 4) THEN
	o_openBuffer := NOT useRequest;
	IF ton_10ms_SettledIncline.Q THEN
		D[900 + mySeq] := 5;
	END_IF;
END_IF;

//Move Bag up incline
ctu_moveUpIncline(CU:=(step = 5) AND NOT Std.HaltSysZone[myZone] AND Std.Clock1s, RESET := (step <> 5), PV := moveUpInclineTime);
IF (step = 5) THEN
	o_openBuffer 	:= (ctu_moveUpIncline.CV <= 4) AND NOT useRequest;//Close buffer stop after 3 seconds running..
	o_runMotor 		:= TRUE;
	IF ctu_moveUpIncline.Q THEN
		D[900 + mySeq] := 6;
	ELSIF NOT Std.HaltSysZone[myZone] THEN
		alarm.Name := ALM_SWITCH_FAULT;
	END_IF;

END_IF;

//Check for line space.
IF (step = 6) THEN
	releaseValid := (NOT i_bagAtBufferOut AND NOT i_bufferOutOpen AND NOT i_BagReleased AND ((myBag = 0) OR ((bag.Cat > 0) AND (bag_out.Cat = 0))));
	IF (myRelLine > 0) THEN
		IF (line_release.Clear AND releaseValid) THEN
			C[myRelLine] := 0;
			D[900 + mySeq] := 7;
		END_IF;
		IF (line_release.Clear AND i_bagAtBufferOut) THEN
			alarm.Name := ALM_SWITCH_FAULT;
		ELSIF (myBag > 0) AND (bag.Cat = 0) THEN
			alarm.Name := ALM_BAG_DATA_ERROR;
			alarm.Time := 0;
		ELSIF line_release.Clear AND (myOutBag > 0) AND (bag_out.Cat > 0) THEN
			alarm.Name := ALM_BAG_DATA_ERROR;
			alarm.Bag := myOutBag;
			alarm.Time := 0;
		END_IF;
	ELSE
		RequestRel.IC[myIC] := releaseValid;
		IF EnableRel.IC[myIC] AND releaseValid THEN

			D[900 + mySeq] := 7;
		ELSIF (myBag > 0) AND (bag.Cat = 0) THEN
			alarm.Name := ALM_BAG_DATA_ERROR;
			alarm.Time := 0;
		ELSIF (myOutBag > 0) AND (bag_out.Cat > 0) THEN
			alarm.Name := ALM_BAG_DATA_ERROR;
			alarm.Bag := myOutBag;
			alarm.Time := 0;
		END_IF;
	END_IF;
	IF i_BagReleased THEN
		alarm.Name := ALM_SWITCH_FAULT;
		alarm.Time := 0;
	END_IF;
	releaseValid := 0; //Clear this as we are using it as a latch in line 7
END_IF;

//Run motor to release bag.
IF (step = 7) THEN
	IF (NOT i_bagAtBufferOut AND NOT i_bufferOutOpen AND ((myBag = 0) OR ((bag.Cat > 0) AND (bag_out.Cat = 0)))) THEN
		releaseValid := 1;
	END_IF;
	o_runMotor := releaseValid AND NOT Std.HaltSysZone[myZone];
	IF releaseValid THEN
		IF (myBag = 0) THEN
			IF (myRelLine > 0) THEN
				IF line_release.Trip THEN
					D[900 + mySeq] := 1;
				END_IF;
			ELSE
				IF NOT EnableRel.IC[myIC] OR i_BagReleased THEN
					D[900 + mySeq] := 1;
				END_IF;
			END_IF;
			IF NOT Std.HaltSysZone[myZone] THEN
				alarm.Name := ALM_BAG_NOT_RELEASED;
			END_IF;
		ELSE//Use tracking
			IF (myRelLine > 0) THEN
				IF line_release.Trip THEN
					bag_out := bag;
					bag := Bag[0];
					D[900 + mySeq] := 1;
				END_IF;
			ELSE
				IF (i_BagReleased OR NOT EnableRel.IC[myIC]) AND (bag.Cat = 0)  THEN // Make sure data is copied out by enabling sequence.
					D[900 + mySeq] := 1;
				ELSIF NOT EnableRel.IC[myIC] AND (bag.Cat > 0) THEN
					alarm.Name := ALM_BAG_DATA_ERROR;
				END_IF;
			END_IF;
		END_IF;
	ELSIF i_bagAtBufferOut OR i_bufferOutOpen THEN
			alarm.Name := ALM_SWITCH_FAULT;
			alarm.Time := 0;
	ELSIF (myBag > 0) THEN
		IF (bag.Cat = 0) THEN
			alarm.Name := ALM_BAG_DATA_ERROR;
			alarm.Time := 0;
		ELSIF (bag_out.Cat > 0) THEN
			alarm.Name := ALM_BAG_DATA_ERROR;
			alarm.Bag := myOutBag;
			alarm.Time := 0;
		END_IF;
	END_IF;
END_IF;

//-----------------------------------
//PLC Outputs - adjust TO suit system
//-----------------------------------

Y[11].Y15	:= o_runMotor;
Y[4].Y16 := o_openBuffer;

//Alarms
timerAlarm(IN := NOT pls AND (alarm.Name > 0),PT:= alarm.Time);

alarm.On 	:= timerAlarm.Q;
alarm.ET 	:= timerAlarm.ET;;

END_PROGRAM
```

### Program Logical/Sequences/10ms/3_clu_2 (IEC) - * Loading unit SLU1

#### 3_slu_1.var
```iecst
VAR RETAIN
	STEP : UINT;
	PLS : BOOL;
	LASTSTEP : UINT;
	EBagSettled : BOOL;
	EBagSettledET : TIME;
	O_OpenStop : BOOL;
	O_SteadyCylinders : BOOL;
	LoadingUnitClear : BOOL;
	LoadingUnitClearET : TIME;
END_VAR
VAR
	CompressCount : UINT;
	O_MoveCompressorUp : BOOL;
	SteadysUpET : TIME;
	SteadysUp : BOOL;
	SteadysDown : BOOL;
	SteadysDownET : TIME;
	I_BagAtBuffer : BOOL;
	O_OpenBufferStop : BOOL;
	I_BagInLoadingUnit : BOOL;
	I_BagFrontPast : BOOL;
	SwitchFault : BOOL;
	TimerAlarm : TON_10ms;
	I_CompressorAtTop : BOOL;
	I_CompressorAtBot : BOOL;
	I_CompressorAtMid : BOOL;
	O_MoveCompressorDn : BOOL;
	BagSettledBuffer : BOOL;
	BagSettledBufferET : TIME;
	I_BagAtSVC1Buffer : BOOL;
	O_SVC1BufferOpen : BOOL;
	I_ChuteBlocked : BOOL;
	CompressorDn : BOOL;
	CompressorDnET : UDINT;
	O_MoveDownTop : BOOL;
	O_MoveDownBottom : BOOL;
	CompressorUp : BOOL;
	CompressorUpET : UDINT;
	O_ElephantsFoot : BOOL;
	I_BagOutCLU2 : BOOL;
END_VAR
```

#### 3_slu_1Cyclic.ab
```automation-basic
PROGRAM _CYCLIC
	(* cyclic program *)

;--------------------------------
;Sequence 3 - Loading Unit D[903]
;--------------------------------

;Inputs / Ouputs

;I_BagOutLoadingUnit     = X904
;I_BagSLU1Trip			= X903
;I_BaginLoadingUnit		= X902

EnableRel.TransferBelt[1]	= FALSE
Request.LU[1]                      = FALSE
;Request.SP[7]                      = FALSE

I_BagAtBuffer			= X[3].X08
I_BagFrontPast		  = X[3].X09
I_BagInLoadingUnit	= X[3].X10
I_BagOutCLU2          = X[3].X11

O_MoveCompressorUp		= FALSE
O_MoveCompressorDn		= FALSE

I_BagAtSVC1Buffer		= FALSE ;X[12].X11
O_SVC1BufferOpen		= FALSE ;Y[12].Y11

O_OpenBufferStop		= FALSE
O_SteadyCylinders		= FALSE
O_OpenStop	 			= FALSE

RequestRel.LU[1]		= FALSE;
Alarm[32].Name 			= 0
Alarm[32].Bag			= 161
Alarm[32].Beacon			= FALSE
Alarm[32].Extra			= 0
Alarm[32].Time			= 3000

;Setup Sequence
;--------------
STEP = D[932]
;Setup Pulse contact
PLS = (STEP <> LASTSTEP)
LASTSTEP = STEP

IF (STEP = 0) THEN
	;Disabled
ENDIF

;Wait for Empty bag at buffer
SwitchFault = ((STEP = 1) AND (I_BagFrontPast OR I_BagInLoadingUnit))
TON_10ms(NOT SwitchFault,200,LoadingUnitClear,LoadingUnitClearET)
TON_10ms(I_BagAtBuffer,300,BagSettledBuffer,BagSettledBufferET)
IF (STEP = 1) THEN
	IF BagSettledBuffer AND LoadingUnitClear AND NOT Std.HaltSys THEN
	;IF LoadingUnitClear AND NOT Std.HaltSys THEN
				;Request.SP[7] = TRUE
		;IF Enable.SP[7] THEN
			D[932] = 2
		;ENDIF
	ENDIF
	IF SwitchFault THEN
		Alarm[32].Name = almSwitchFault
	ELSE
		Alarm[32].Name = almNoAlarm
	ENDIF
ENDIF

;Open stops let bag in Loading Unit
IF (STEP = 2) THEN
	O_OpenStop 			= TRUE
	O_OpenBufferStop 	= TRUE
	;Enable.LU[1]		= NOT I_BagFrontPast
	IF I_BagFrontPast THEN
		D[932] = 3
	ENDIF
	Alarm[32].Name = almBagNotArrived
ENDIF

;Wait for bag to settle
TON_10ms(I_BagInLoadingUnit,300,EBagSettled,EBagSettledET)
IF (STEP = 3) THEN
	IF EBagSettled THEN
		D[932] = 4
	ENDIF
	Alarm[32].Name = almBagNotSettled
	;Special for Banbury - SVC1 is also a loading hoist
	;IF SVC1RequestEmpty THEN
	;	Bag[221].Cat 	= 99
	;	D[903] 			= 9
	;ENDIF
ENDIF

;Steady cylinders on from steps 4 - 5
O_SteadyCylinders = ((STEP = 4) OR (STEP = 5))

;Move Steady Cylinders down
TON_10ms((STEP = 4),300,SteadysDown,SteadysDownET)
IF (STEP = 4) THEN
	IF (SteadysDown AND (Bag[161].Cat = 0)) THEN
		D[932] = 5
	ENDIF
	IF (Bag[161].Cat <> 0) THEN
		Alarm[32].Name = almBagDataError
	ELSE
		Alarm[32].Name = almNoAlarm
	ENDIF
ENDIF

;Wait for bag to be loaded
IF (STEP = 5) THEN
	EnableRel.TransferBelt[1] = TRUE
	IF (Bag[161].Cat > 0) THEN
		D[932] = 6
	ENDIF
	Alarm[32].Name = almNoAlarm ;Transfer belt should alarm
ENDIF

;Allow Steady Cylinders to move up
TON_10ms((STEP = 6),300,SteadysUp,SteadysUpET)
IF (STEP = 6) THEN
	IF SteadysUp AND NOT Enable.LU[1] THEN

			D[932] = 7

	ENDIF
	IF Enable.LU[1] THEN
		Alarm[32].Name = almReceiveSwitchFault
	ENDIF
ENDIF

;

;Check for space at Buffer
TON_10ms((STEP = 7),300,SteadysUp,SteadysUpET)
IF (STEP = 7) THEN
	IF NOT Std.HaltSys AND SteadysUp AND (Bag[221].Cat = 0) THEN
		Request.LU[1] = TRUE
		IF Enable.LU[1] THEN
			IF (Bag[161].Cat>0) AND (Bag[164].Cat = 0) THEN
							Bag[164] = Bag[161]
							Bag[161] = Bag[0]
			ENDIF
			;C[34]   = 0
			D[932] 	= 8
			;ELSE
			;Alarm[3].Name = almSwitchFault
		ENDIF
		;ENDIF
	ENDIF
ENDIF

;Open stop - Unitl bag out
IF (STEP = 8) THEN
	O_OpenStop = TRUE
	;IF PLS THEN
	;	C[16] = 0
	;ENDIF
	;IF Line[16].Trip THEN
	IF I_BagOutCLU2  THEN

		D[932] = 1
	ENDIF
	Alarm[32].Name = almBagNotReleased
ENDIF

;Alarms
TimerAlarm.IN = NOT PLS AND (Alarm[32].Name > 0)
TimerAlarm.PT = Alarm[32].Time
TimerAlarm FUB TON_10ms()
Alarm[32].On = TimerAlarm.Q
Alarm[32].ET = TimerAlarm.ET

;Outputs
;-------

Y[3].Y06 = O_OpenBufferStop
Y[3].Y08 = O_SteadyCylinders
Y[3].Y09 = O_OpenStop

;Y[8].Y10 = O_MoveDownTop
;Y[8].Y09 = O_MoveDownBottom
;Y[8].Y15 = O_ElephantsFoot
END_PROGRAM
```

### Program Logical/Sequences/10ms/20_cp17 (IEC) - * SP2 Empty bags from SDC1/2

#### 12_sp2.var
```iecst
VAR RETAIN
	STEP : UINT;
	PLS : BOOL;
	LASTSTEP : UINT;
END_VAR
VAR
	TimerAlarm : TON_10ms;
	I_BagAtBuffer : ARRAY[0..5] OF BOOL;
	O_OpenBuffer : BOOL;
	SDC2BufferFullET : TIME;
	SDC2BufferFull : BOOL;
	SettledBufferET : TIME;
	SettledBuffer : ARRAY[0..2] OF BOOL;
	O_OpenSP2BufferStop : BOOL;
	O_SelectPoint : BOOL;
	SP2BufferFull : BOOL;
	SP2BufferFullET : UDINT;
	ParingLoopEnabled : BOOL;
	BagInLoopHasDest : BOOL;
	BagAtBuffer : ARRAY[0..5] OF BOOL;
	SettledBufferSVC1 : BOOL;
	SettledBufferSVC1ET : UDINT;
	SettledBufferSVC2 : BOOL;
	SettledBufferSVC2ET : UDINT;
	O_SelectPointSVC1 : BOOL;
	O_SelectPointSVC2 : BOOL;
	Reset : BOOL;
	ResetET : UDINT;
	I_BagatBuffer : BOOL;
	BagAtBufferET : ARRAY[0..5] OF UDINT;
	Alernate : USINT;
	I_BagAtSVC1BufferStop : BOOL;
	O_SVC1BufferStop : BOOL;
	I_BagAtSVC2BufferStop : BOOL;
	O_SVC2BufferStop : BOOL;
	O_SelectSVC1 : BOOL;
	O_SelectSVC2 : BOOL;
	MySeq : USINT;
	MyBag : USINT;
	O_SelectCDC9 : BOOL;
	O_SelectCPI6 : BOOL;
	O_SelectCDC4 : BOOL;
	O_SelectStraight : BOOL;
	BagSettledBufferET : ARRAY[0..2] OF UDINT;
	Alt : USINT;
	O_SelectCLU1 : BOOL;
	O_SelectCLU2 : BOOL;
END_VAR
```

#### 12_sp2Cyclic.ab
```automation-basic
PROGRAM _CYCLIC
	(* cyclic program *)

;---------------------------------------
;Sequence 8 - SP8 Single point 2 D[912]
;---------------------------------------

;Inputs

I_BagAtBuffer[1]		= Request.LU[1]
I_BagAtBuffer[2]		= Request.LU[2]

MySeq                   = 20

Alarm[MySeq].Name 			= 0
Alarm[MySeq].Bag			= 164
Alarm[MySeq].Beacon		= TRUE
Alarm[MySeq].Extra			= 0
Alarm[MySeq].Time			= 1500

O_SelectCLU1                = FALSE
O_SelectCLU2                = FALSE
Enable.LU[1]                = FALSE
Enable.LU[2]                = FALSE

;Setup Sequence
STEP = D[900 + MySeq]
;Setup Pulse contact
PLS = (STEP <> LASTSTEP)
LASTSTEP = STEP

;Sequence
;Step 0 - Disabled
IF (STEP = 0) THEN
	;Disabled
ENDIF

;reset points
TON_10ms((STEP = 1),200,Reset,ResetET)
IF (STEP = 1) THEN

	IF (Line[9].Clear)  THEN
		D[900 + MySeq] = 2
	ENDIF
	ELSE

ENDIF

;check which bag is ready
TON_10ms(I_BagAtBuffer[1],200,SettledBuffer[1],BagSettledBufferET[1])
TON_10ms(I_BagAtBuffer[2],200,SettledBuffer[2],BagSettledBufferET[2])
IF (STEP = 2) THEN
	IF (Line[9].Clear) THEN
		Alt = Alt + 1
		IF (Alt > 2) THEN
			Alt = 0
		ENDIF
		IF SettledBuffer[1] AND (Alt = 1) THEN
			C[9]          = 0
		    D[900 + MySeq] = 3
		ELSE IF SettledBuffer[2] AND (Alt = 2) THEN
			C[9]          = 0
			D[900 + MySeq] = 4
		ENDIF
	ENDIF
ENDIF

;Bag at line
IF (STEP = 3) THEN
	O_SelectCLU1  = TRUE
	Enable.LU[1]  = TRUE
	IF (Line[9].Trip = TRUE) THEN
		IF (Bag[164].Cat > 0) AND (Bag[118].Cat = 0) THEN
			IF (Bag[164].Dst >6) AND (Bag[164].Dst <>14) THEN
				Bag[164].Dst = 0
			ENDIF
			Bag[118] = Bag[164]
			Bag[164] = Bag[0]
		ENDIF
		D[900 + MySeq] = 1
	ENDIF
	Alarm[MySeq].Name 	  = almBagNotArrived
ENDIF

;Bag at line
IF (STEP = 4) THEN
	O_SelectCLU2 = TRUE
	Enable.LU[2]  = TRUE
	IF (Line[9].Trip = TRUE) THEN
		IF (Bag[164].Cat > 0) AND (Bag[118].Cat = 0) THEN
		     IF (Bag[164].Dst >6) AND (Bag[164].Dst <>14) THEN
				Bag[164].Dst = 0
			ENDIF
			Bag[118] = Bag[164]
			Bag[164] = Bag[0]
		ENDIF
		D[900 + MySeq] = 1
	ENDIF
	Alarm[MySeq].Name 	  = almBagNotArrived
ENDIF

;Alarms
TimerAlarm.IN 	= NOT PLS AND (Alarm[MySeq].Name > 0)
TimerAlarm.PT 	= Alarm[MySeq].Time
TimerAlarm FUB TON_10ms()
Alarm[MySeq].On 	= TimerAlarm.Q
Alarm[MySeq].ET 	= TimerAlarm.ET

;Outputs
Y[3].Y11 = O_SelectCLU2
Y[3].Y10 = O_SelectCLU1
END_PROGRAM
```

### Program Logical/Sequences/10ms/21_cpi1 (IEC) - *Pneumatic Incline

#### pic.var
```iecst
(********************************************************************
 * COPYRIGHT --
 ********************************************************************
 * Program: pr
 * File: pr.var
 * Author: treamsbottom
 * Created: July 16, 2015
 ********************************************************************
 * Local variables of program pr
 ********************************************************************)
VAR
	mySeq : UINT;
	myIO : UINT;
	myZone : UINT;
	myRelLine : UINT;
	myBag : UINT;
	i_bagAtBuffer : BOOL;
	i_bagAtBufferOut : BOOL;
	i_bufferOutOpen : BOOL;
	o_openBuffer : BOOL;
	step : UINT;
	pls : BOOL;
	timerAlarm : TON_10ms;
END_VAR
VAR RETAIN
	lastStep : UINT;
END_VAR
VAR
	bufferSettleTime : UDINT;
	myOutBag : UINT;
	myBuffBag : UINT;
	myPI : UINT;
	i_bagInIncline : BOOL;
	i_cylinderAtBottom : BOOL;
	i_cylinderAtTop : BOOL;
	o_cylinderDown : BOOL;
	useRequest : BOOL;
	releaseValid : BOOL;
	ton_10ms_SettledBuffer : TON_10ms;
	ton_10ms_SettledInIncline : TON_10ms;
	ton_10ms_CylinderDown : TON_10ms;
	kev : BOOL;
END_VAR
```

#### pic.st
```iecst
(********************************************************************
 * COPYRIGHT --
 ********************************************************************
 * Program: pic
 * File: pic.st
 * Author: treamsbottom
 * Created: July 16, 2015
 ********************************************************************
 * Implementation of program pic - Pneumatic Incline
 ********************************************************************)
//V1.00.1 First Release
PROGRAM _INIT
//Configuration
mySeq						:= 21;	//Sequence number
myIO						:= 7;
myZone						:= 0;
myRelLine					:= 28;
myBuffBag					:= 0;
myBag						:= 0;
bufferSettleTime			:= 300;
myPI						:= 1;

myOutBag 					:= Line[myRelLine].LastBag;
END_PROGRAM

PROGRAM _CYCLIC
//Inputs

i_bagInIncline			:= X[myIO].X10;
i_cylinderAtBottom		:= X[myIO].X12;
i_cylinderAtTop			:= X[myIO].X11;
i_bagAtBuffer			:= X[myIO].X09;

i_bagAtBufferOut 		:= FALSE; // Any Single bag buffer out IO.
i_bufferOutOpen			:= FALSE;

o_openBuffer			:= FALSE;
o_cylinderDown			:= FALSE;

Request.PI[myPI]		:= FALSE;
RequestRel.PI[myPI]		:= FALSE;

IF (myBag = 0) THEN
//	Alarm[mySeq].Bag	:= 10014;
ELSE
//	Alarm[mySeq].Bag	:= myBag;
END_IF;

Alarm[mySeq].Name 		:= 0;
Alarm[mySeq].Beacon	:= TRUE;
Alarm[mySeq].Bag	:= 10014;
Alarm[mySeq].Extra		:= 0;
Alarm[mySeq].Time		:= 3000;

//Setup Sequence
step := D[900 + mySeq];
//Setup Pulse contact
pls := (step <> lastStep);
lastStep := step;

//Sequence
IF (step = 0) THEN
	//Disabled
END_IF;

//Wait for at buffer
ton_10ms_SettledBuffer(IN:= i_bagAtBuffer, PT:= bufferSettleTime);
IF (step = 1) THEN
	IF NOT Std.HaltSysZone[myZone] AND i_cylinderAtTop AND NOT i_bagInIncline THEN
		IF useRequest THEN
			D[900 + mySeq] := 2;
		ELSE
			IF ton_10ms_SettledBuffer.Q THEN
				IF (myBuffBag > 0) THEN
					IF (Bag[myBuffBag].Cat > 0) AND (Bag[myBag].Cat = 0) THEN
						D[900 + mySeq] := 2;
					ELSIF (Bag[myBuffBag].Cat = 0) THEN
						Alarm[mySeq].Name := ALM_BAG_DATA_ERROR;
						Alarm[mySeq].Bag := myBuffBag;
					ELSE
						Alarm[mySeq].Name := ALM_BAG_DATA_ERROR;
					END_IF;
				ELSE
					D[900 + mySeq] := 2;
				END_IF;
			ELSIF (myBuffBag > 0) AND (Bag[myBuffBag].Cat > 0) THEN
				Alarm[mySeq].Name := ALM_BAG_NOT_SETTLED;
			END_IF;
		END_IF;
	ELSIF NOT Std.HaltSysZone[myZone] THEN
		Alarm[mySeq].Name := ALM_SWITCH_FAULT;
	END_IF;

END_IF;

//Open Buffer stop
IF (step = 2) THEN
	releaseValid := ((myBag = 0) OR ((Bag[myBag].Cat = 0) AND (Bag[myBuffBag].Cat > 0)));
	o_openBuffer	   := releaseValid AND NOT useRequest;
	Request.PI[myPI]  := releaseValid AND useRequest;
	IF (i_bagInIncline AND releaseValid) THEN
		IF (myBag > 0) THEN
			Bag[myBag] := Bag[myBuffBag]; //Clear empty buffer bag data if used
			Bag[myBuffBag] := Bag[0];
		END_IF;
		D[900 + mySeq] := 3;
	ELSIF (myBag > 0) THEN
		IF (Bag[myBag].Cat > 0) THEN
			Alarm[mySeq].Name := ALM_BAG_DATA_ERROR;
			Alarm[mySeq].Time := 0;
		ELSIF (Bag[myBuffBag].Cat = 0) THEN
			Alarm[mySeq].Name := ALM_BAG_DATA_ERROR;
			Alarm[mySeq].Bag := myBuffBag;
			Alarm[mySeq].Time := 0;
		ELSE
			Alarm[mySeq].Name  := ALM_BAG_NOT_ARRIVED;
		END_IF;
		Alarm[mySeq].Name  := ALM_BAG_NOT_ARRIVED;
	END_IF;
END_IF;

//Let bag settle at base OF incline
ton_10ms_SettledInIncline(IN:= i_bagInIncline, PT:= 300);
IF (step = 3) THEN
	o_openBuffer := NOT useRequest;
	IF  ton_10ms_SettledInIncline.Q AND NOT Std.HaltSysZone[myZone] THEN
		D[900 + mySeq] := 4;
	ELSIF NOT Std.HaltSysZone[myZone] THEN
		Alarm[mySeq].Name := ALM_BAG_NOT_SETTLED;
	END_IF;
END_IF

//Move incline down to collect first trolley
ton_10ms_CylinderDown(IN := i_cylinderAtBottom, PT:=300);
IF (step = 4) THEN
	o_openBuffer := NOT useRequest;
	o_cylinderDown := TRUE;
	IF ton_10ms_CylinderDown.Q THEN
		D[900 + mySeq] := 5;
	END_IF;
	Alarm[mySeq].Name := ALM_SWITCH_FAULT;
END_IF;

//Let cylinder move back to the top.
IF (step = 5) THEN
	o_openBuffer := NOT useRequest;
	IF i_cylinderAtTop THEN
		D[900 + mySeq] := 6;
	END_IF;
	Alarm[mySeq].Name := ALM_SWITCH_FAULT;
END_IF;

//Check for valid release..
//Check for line space.
IF (step = 6) THEN
	releaseValid := ( NOT i_cylinderAtBottom AND NOT i_bagAtBufferOut AND NOT i_bufferOutOpen AND ((myBag = 0) OR ((Bag[myBag].Cat > 0) AND (Bag[myOutBag].Cat = 0))));
	IF (myRelLine > 0) THEN
		IF (Line[myRelLine].Clear AND releaseValid) THEN
			C[myRelLine] := 0;
			D[900 + mySeq] := 7;
		END_IF;
		IF i_cylinderAtBottom OR NOT i_bagInIncline THEN
			Alarm[mySeq].Name := ALM_SWITCH_FAULT;
			Alarm[mySeq].Time := 0;
		ELSIF (Line[myRelLine].Clear AND i_bagAtBufferOut) THEN
			Alarm[mySeq].Name := ALM_SWITCH_FAULT;
		ELSIF (myBag > 0) AND (Bag[myBag].Cat = 0) THEN
			Alarm[mySeq].Name := ALM_BAG_DATA_ERROR;
			Alarm[mySeq].Time := 0;
		ELSIF Line[myRelLine].Clear AND (myOutBag > 0) AND (Bag[myOutBag].Cat > 0) THEN
			Alarm[mySeq].Name := ALM_BAG_DATA_ERROR;
			Alarm[mySeq].Bag := myOutBag;
			Alarm[mySeq].Time := 0;
		END_IF;
	ELSE
		RequestRel.PI[myPI] := releaseValid;
		IF EnableRel.PI[myPI] AND releaseValid THEN
			D[900 + mySeq] := 7;
		ELSIF NOT i_cylinderAtBottom OR NOT i_bagInIncline THEN
			Alarm[mySeq].Name := ALM_SWITCH_FAULT;
			Alarm[mySeq].Time := 0;
		ELSIF (myBag > 0) AND (Bag[myBag].Cat = 0) THEN
			Alarm[mySeq].Name := ALM_BAG_DATA_ERROR;
			Alarm[mySeq].Time := 0;
		ELSIF (myOutBag > 0) AND (Bag[myOutBag].Cat > 0) THEN
			Alarm[mySeq].Name := ALM_BAG_DATA_ERROR;
			Alarm[mySeq].Bag := myOutBag;
			Alarm[mySeq].Time := 0;
		END_IF;
	END_IF;
END_IF;

//Move cylinder down to get 2nd trolley.
IF (step = 7) THEN
	o_cylinderDown := TRUE;
	IF  ton_10ms_CylinderDown.Q THEN
		D[900 + mySeq] := 8;
	END_IF;
	Alarm[mySeq].Name := ALM_SWITCH_FAULT;
END_IF;

//Release bag
IF (step = 8) THEN
	releaseValid := (NOT i_bagAtBufferOut AND NOT i_bufferOutOpen AND ((myBag = 0) OR ((Bag[myBag].Cat > 0) AND (Bag[myOutBag].Cat = 0))));
	o_cylinderDown := NOT releaseValid; // Hold cylinder down if release is not valid.
	IF releaseValid THEN
		IF (myBag = 0) THEN// Not tracking.
			IF (myRelLine > 0) THEN
				IF Line[myRelLine].Trip THEN
					D[900 + mySeq] := 1;
				END_IF;
			ELSE
				IF NOT EnableRel.PI[myPI] THEN
					D[900 + mySeq] := 1;
				END_IF;
			END_IF;
			IF NOT Std.HaltSysZone[myZone] THEN
				Alarm[mySeq].Name := ALM_BAG_NOT_RELEASED;
			END_IF;
		ELSE//Use tracking
			IF (myRelLine > 0) THEN
				IF Line[myRelLine].Trip THEN
					Bag[myOutBag] := Bag[myBag];
					Bag[myBag] := Bag[0];
					D[900 + mySeq] := 1;
				END_IF;
			ELSE
				IF NOT EnableRel.PI[myPI] AND (Bag[myBag].Cat = 0) THEN // Make sure data is copied out by enabling sequence.
					D[900 + mySeq] := 1;
				ELSIF NOT EnableRel.PI[myPI] AND (Bag[myBag].Cat > 0) THEN
					Alarm[mySeq].Name := ALM_BAG_DATA_ERROR;
				END_IF;
			END_IF;
		END_IF;
	ELSIF i_bagAtBufferOut AND NOT i_bufferOutOpen THEN
		Alarm[mySeq].Name := ALM_SWITCH_FAULT;
		Alarm[mySeq].Time := 0;
	ELSIF (myBag > 0) THEN
		IF (Bag[myBag].Cat = 0) THEN
			Alarm[mySeq].Name := ALM_BAG_DATA_ERROR;
			Alarm[mySeq].Time := 0;
		ELSIF (Bag[myOutBag].Cat > 0) THEN
			Alarm[mySeq].Name := ALM_BAG_DATA_ERROR;
			Alarm[mySeq].Bag := myOutBag;
			Alarm[mySeq].Time := 0;
		END_IF;
	END_IF;
END_IF

//-----------------------------------
//PLC Outputs - adjust TO suit system
//-----------------------------------
kev := o_cylinderDown;
Y[11].Y07 := o_cylinderDown;
Y[3].Y13 := o_openBuffer;

//Alarms
timerAlarm(IN := NOT pls AND (Alarm[mySeq].Name > 0),PT:= Alarm[mySeq].Time);

Alarm[mySeq].On 	:= timerAlarm.Q;
Alarm[mySeq].ET 	:= timerAlarm.ET;

END_PROGRAM
```

### Program Logical/Sequences/10ms/22_cpi2 (IEC) - *Pneumatic Incline

#### pic.st
```iecst
(********************************************************************
 * COPYRIGHT --
 ********************************************************************
 * Program: pic
 * File: pic.st
 * Author: treamsbottom
 * Created: July 16, 2015
 ********************************************************************
 * Implementation of program pic - Pneumatic Incline
 ********************************************************************)
//V1.00.1 First Release
PROGRAM _INIT
//Configuration
mySeq						:= 22;	//Sequence number
myIO						:= 7;
myZone						:= 0;
myRelLine					:= 38;
myBuffBag					:= 0;
myBag						:= 0;
bufferSettleTime			:= 300;
myPI						:= 2;

myOutBag 					:= Line[myRelLine].LastBag;
END_PROGRAM

PROGRAM _CYCLIC
//Inputs

i_bagInIncline			:= X[7].X15;
i_cylinderAtBottom		:= X[8].X01;
i_cylinderAtTop			:= X[7].X16;
i_bagAtBuffer			:= X[7].X14;

i_bagAtBufferOut 		:= FALSE; // Any Single bag buffer out IO.
i_bufferOutOpen			:= FALSE;

o_openBuffer			:= FALSE;
o_cylinderDown			:= FALSE;

Request.PI[myPI]		:= FALSE;
RequestRel.PI[myPI]		:= FALSE;

IF (myBag = 0) THEN
	Alarm[mySeq].Bag	:= 10016;
ELSE
//	Alarm[mySeq].Bag	:= myBag;
END_IF;

Alarm[mySeq].Name 		:= 0;
Alarm[mySeq].Bag	:= 10016;
Alarm[mySeq].Beacon	:= TRUE;
Alarm[mySeq].Extra		:= 0;
Alarm[mySeq].Time		:= 3000;

//Setup Sequence
step := D[900 + mySeq];
//Setup Pulse contact
pls := (step <> lastStep);
lastStep := step;

//Sequence
IF (step = 0) THEN
	//Disabled
END_IF;

//Wait for at buffer
ton_10ms_SettledBuffer(IN:= i_bagAtBuffer, PT:= bufferSettleTime);
IF (step = 1) THEN
	IF NOT Std.HaltSysZone[myZone] AND i_cylinderAtTop AND NOT i_bagInIncline THEN
		IF useRequest THEN
			D[900 + mySeq] := 2;
		ELSE
			IF ton_10ms_SettledBuffer.Q THEN
				IF (myBuffBag > 0) THEN
					IF (Bag[myBuffBag].Cat > 0) AND (Bag[myBag].Cat = 0) THEN
						D[900 + mySeq] := 2;
					ELSIF (Bag[myBuffBag].Cat = 0) THEN
						Alarm[mySeq].Name := ALM_BAG_DATA_ERROR;
						Alarm[mySeq].Bag := myBuffBag;
					ELSE
						Alarm[mySeq].Name := ALM_BAG_DATA_ERROR;
					END_IF;
				ELSE
					D[900 + mySeq] := 2;
				END_IF;
			ELSIF (myBuffBag > 0) AND (Bag[myBuffBag].Cat > 0) THEN
				Alarm[mySeq].Name := ALM_BAG_NOT_SETTLED;
			END_IF;
		END_IF;
	ELSIF NOT Std.HaltSysZone[myZone] THEN
		Alarm[mySeq].Name := ALM_SWITCH_FAULT;
	END_IF;
END_IF;

//Open Buffer stop
IF (step = 2) THEN
	releaseValid := ((myBag = 0) OR ((Bag[myBag].Cat = 0) AND (Bag[myBuffBag].Cat > 0)));
	o_openBuffer	   := releaseValid AND NOT useRequest;
	Request.PI[myPI]  := releaseValid AND useRequest;
	IF (i_bagInIncline AND releaseValid) THEN
		IF (myBag > 0) THEN
			Bag[myBag] := Bag[myBuffBag]; //Clear empty buffer bag data if used
			Bag[myBuffBag] := Bag[0];
		END_IF;
		D[900 + mySeq] := 3;
	ELSIF (myBag > 0) THEN
		IF (Bag[myBag].Cat > 0) THEN
			Alarm[mySeq].Name := ALM_BAG_DATA_ERROR;
			Alarm[mySeq].Time := 0;
		ELSIF (Bag[myBuffBag].Cat = 0) THEN
			Alarm[mySeq].Name := ALM_BAG_DATA_ERROR;
			Alarm[mySeq].Bag := myBuffBag;
			Alarm[mySeq].Time := 0;
		ELSE
			Alarm[mySeq].Name  := ALM_BAG_NOT_ARRIVED;
		END_IF;
		Alarm[mySeq].Name  := ALM_BAG_NOT_ARRIVED;
	END_IF;
END_IF;

//Let bag settle at base OF incline
ton_10ms_SettledInIncline(IN:= i_bagInIncline, PT:= 300);
IF (step = 3) THEN
	o_openBuffer := NOT useRequest;
	IF  ton_10ms_SettledInIncline.Q AND NOT Std.HaltSysZone[myZone] THEN
		D[900 + mySeq] := 4;
	ELSIF NOT Std.HaltSysZone[myZone] THEN
		Alarm[mySeq].Name := ALM_BAG_NOT_SETTLED;
	END_IF;
END_IF

//Move incline down to collect first trolley
ton_10ms_CylinderDown(IN := i_cylinderAtBottom, PT:=300);
IF (step = 4) THEN
	o_openBuffer := NOT useRequest;
	o_cylinderDown := TRUE;
	IF ton_10ms_CylinderDown.Q THEN
		D[900 + mySeq] := 5;
	END_IF;
	Alarm[mySeq].Name := ALM_SWITCH_FAULT;
END_IF;

//Let cylinder move back to the top.
IF (step = 5) THEN
	o_openBuffer := NOT useRequest;
	IF i_cylinderAtTop THEN
		D[900 + mySeq] := 6;
	END_IF;
	Alarm[mySeq].Name := ALM_SWITCH_FAULT;
END_IF;

//Check for valid release..
//Check for line space.
IF (step = 6) THEN
	releaseValid := (ton_10ms_SettledInIncline.Q AND NOT i_cylinderAtBottom AND NOT i_bagAtBufferOut AND NOT i_bufferOutOpen AND ((myBag = 0) OR ((Bag[myBag].Cat > 0) AND (Bag[myOutBag].Cat = 0))));
	IF (myRelLine > 0) THEN
		IF (Line[myRelLine].Clear AND releaseValid) THEN
			C[myRelLine] := 0;
			D[900 + mySeq] := 7;
		END_IF;
		IF i_cylinderAtBottom OR NOT i_bagInIncline THEN
			Alarm[mySeq].Name := ALM_SWITCH_FAULT;
			Alarm[mySeq].Time := 0;
		ELSIF (Line[myRelLine].Clear AND i_bagAtBufferOut) THEN
			Alarm[mySeq].Name := ALM_SWITCH_FAULT;
		ELSIF (myBag > 0) AND (Bag[myBag].Cat = 0) THEN
			Alarm[mySeq].Name := ALM_BAG_DATA_ERROR;
			Alarm[mySeq].Time := 0;
		ELSIF Line[myRelLine].Clear AND (myOutBag > 0) AND (Bag[myOutBag].Cat > 0) THEN
			Alarm[mySeq].Name := ALM_BAG_DATA_ERROR;
			Alarm[mySeq].Bag := myOutBag;
			Alarm[mySeq].Time := 0;
		END_IF;
	ELSE
		RequestRel.PI[myPI] := releaseValid;
		IF EnableRel.PI[myPI] AND releaseValid THEN
			D[900 + mySeq] := 7;
		ELSIF NOT i_cylinderAtBottom OR NOT i_bagInIncline THEN
			Alarm[mySeq].Name := ALM_SWITCH_FAULT;
			Alarm[mySeq].Time := 0;
		ELSIF (myBag > 0) AND (Bag[myBag].Cat = 0) THEN
			Alarm[mySeq].Name := ALM_BAG_DATA_ERROR;
			Alarm[mySeq].Time := 0;
		ELSIF (myOutBag > 0) AND (Bag[myOutBag].Cat > 0) THEN
			Alarm[mySeq].Name := ALM_BAG_DATA_ERROR;
			Alarm[mySeq].Bag := myOutBag;
			Alarm[mySeq].Time := 0;
		END_IF;
	END_IF;
END_IF;

//Move cylinder down to get 2nd trolley.
IF (step = 7) THEN
	o_cylinderDown := TRUE;
	IF  ton_10ms_CylinderDown.Q THEN
		D[900 + mySeq] := 8;
	END_IF;
	Alarm[mySeq].Name := ALM_SWITCH_FAULT;
END_IF;

//Release bag
IF (step = 8) THEN
	releaseValid := (NOT i_bagAtBufferOut AND NOT i_bufferOutOpen AND ((myBag = 0) OR ((Bag[myBag].Cat > 0) AND (Bag[myOutBag].Cat = 0))));
	o_cylinderDown := NOT releaseValid; // Hold cylinder down if release is not valid.
	IF releaseValid THEN
		IF (myBag = 0) THEN// Not tracking.
			IF (myRelLine > 0) THEN
				IF Line[myRelLine].Trip THEN
					D[900 + mySeq] := 1;
				END_IF;
			ELSE
				IF NOT EnableRel.PI[myPI] THEN
					D[900 + mySeq] := 1;
				END_IF;
			END_IF;
			IF NOT Std.HaltSysZone[myZone] THEN
				Alarm[mySeq].Name := ALM_BAG_NOT_RELEASED;
			END_IF;
		ELSE//Use tracking
			IF (myRelLine > 0) THEN
				IF Line[myRelLine].Trip THEN
					Bag[myOutBag] := Bag[myBag];
					Bag[myBag] := Bag[0];
					D[900 + mySeq] := 1;
				END_IF;
			ELSE
				IF NOT EnableRel.PI[myPI] AND (Bag[myBag].Cat = 0) THEN // Make sure data is copied out by enabling sequence.
					D[900 + mySeq] := 1;
				ELSIF NOT EnableRel.PI[myPI] AND (Bag[myBag].Cat > 0) THEN
					Alarm[mySeq].Name := ALM_BAG_DATA_ERROR;
				END_IF;
			END_IF;
		END_IF;
	ELSIF i_bagAtBufferOut AND NOT i_bufferOutOpen THEN
		Alarm[mySeq].Name := ALM_SWITCH_FAULT;
		Alarm[mySeq].Time := 0;
	ELSIF (myBag > 0) THEN
		IF (Bag[myBag].Cat = 0) THEN
			Alarm[mySeq].Name := ALM_BAG_DATA_ERROR;
			Alarm[mySeq].Time := 0;
		ELSIF (Bag[myOutBag].Cat > 0) THEN
			Alarm[mySeq].Name := ALM_BAG_DATA_ERROR;
			Alarm[mySeq].Bag := myOutBag;
			Alarm[mySeq].Time := 0;
		END_IF;
	END_IF;
END_IF

//-----------------------------------
//PLC Outputs - adjust TO suit system
//-----------------------------------

Y[11].Y08 := o_cylinderDown;
Y[3].Y14 := o_openBuffer;

//Alarms
timerAlarm(IN := NOT pls AND (Alarm[mySeq].Name > 0),PT:= Alarm[mySeq].Time);

Alarm[mySeq].On 	:= timerAlarm.Q;
Alarm[mySeq].ET 	:= timerAlarm.ET;

END_PROGRAM
```

### Program Logical/Sequences/10ms/23_cpi3 (IEC, version 1.00.3) - *Pneumatic Incline
